LIN {X 0.078,Y -589.300,Z 1509.135,A 0.000,B 0.000,C 90.000,E1 60.205} C_DIS
LIN {X 0.071,Y -590.792,Z 1509.123,A 0.000,B 0.000,C 90.000,E1 58.074} C_DIS
LIN {X -0.260,Y -591.564,Z 1509.117,A 0.000,B 0.000,C 90.000,E1 57.041} C_DIS
LIN {X 0.336,Y -592.759,Z 1509.108,A 0.000,B 0.000,C 90.000,E1 55.388} C_DIS
LIN {X 0.156,Y -593.285,Z 1509.104,A 0.000,B 0.000,C 90.000,E1 54.609} C_DIS
LIN {X -0.185,Y -594.026,Z 1509.095,A 0.000,B 0.000,C 90.000,E1 53.050} C_DIS
LIN {X 0.067,Y -594.863,Z 1509.084,A 0.000,B 0.000,C 90.000,E1 51.170} C_DIS
LIN {X 0.249,Y -595.682,Z 1509.074,A 0.000,B 0.000,C 90.000,E1 49.299} C_DIS
LIN {X 0.240,Y -595.941,Z 1509.071,A 0.000,B 0.000,C 90.000,E1 48.771} C_DIS
LIN {X 0.220,Y -596.064,Z 1509.065,A 0.000,B 0.000,C 90.000,E1 47.715} C_DIS
LIN {X -0.242,Y -596.037,Z 1509.059,A 0.000,B 0.000,C 90.000,E1 46.701} C_DIS
LIN {X -0.293,Y -595.880,Z 1509.053,A 0.000,B 0.000,C 90.000,E1 45.648} C_DIS
LIN {X 0.106,Y -595.808,Z 1509.051,A 0.000,B 0.000,C 90.000,E1 45.081} C_DIS
LIN {X -0.170,Y -595.079,Z 1509.043,A 0.000,B 0.000,C 90.000,E1 43.785} C_DIS
LIN {X -0.010,Y -594.518,Z 1509.039,A 0.000,B 0.000,C 90.000,E1 42.975} C_DIS
LIN {X -0.054,Y -593.537,Z 1509.033,A 0.000,B 0.000,C 90.000,E1 41.919} C_DIS
LIN {X -0.103,Y -592.480,Z 1509.027,A 0.000,B 0.000,C 90.000,E1 40.862} C_DIS
LIN {X -0.164,Y -591.177,Z 1509.021,A 0.000,B 0.000,C 90.000,E1 39.806} C_DIS
LIN {X -0.249,Y -589.695,Z 1509.015,A 0.000,B 0.000,C 90.000,E1 38.749} C_DIS
LIN {X 0.097,Y -587.768,Z 1509.009,A 0.000,B 0.000,C 90.000,E1 37.649} C_DIS
LIN {X -0.136,Y -586.038,Z 1509.005,A 0.000,B 0.000,C 90.000,E1 36.870} C_DIS
LIN {X 0.248,Y -584.795,Z 1509.002,A 0.000,B 0.000,C 90.000,E1 36.297} C_DIS
LIN {X -0.195,Y -583.162,Z 1508.999,A 0.000,B 0.000,C 90.000,E1 35.804} C_DIS
LIN {X 0.165,Y -581.111,Z 1508.996,A 0.000,B 0.000,C 90.000,E1 35.231} C_DIS
LIN {X 0.256,Y -579.158,Z 1508.994,A 0.000,B 0.000,C 90.000,E1 34.818} C_DIS
LIN {X 0.092,Y -577.527,Z 1508.992,A 0.000,B 0.000,C 90.000,E1 34.565} C_DIS
LIN {X -0.139,Y -576.519,Z 1508.991,A 0.000,B 0.000,C 90.000,E1 34.452} C_DIS
LIN {X -0.224,Y -575.268,Z 1508.991,A 0.000,B 0.000,C 90.000,E1 34.326} C_DIS
LIN {X -0.308,Y -573.503,Z 1508.990,A 0.000,B 0.000,C 90.000,E1 34.199} C_DIS
LIN {X -0.047,Y -572.090,Z 1508.990,A 0.000,B 0.000,C 90.000,E1 34.119} C_DIS
LIN {X -0.068,Y -397.232,Z 1508.990,A 0.000,B 0.000,C 90.000,E1 34.119} C_DIS
LIN {X 0.195,Y -393.782,Z 1508.977,A 0.000,B 0.000,C 90.000,E1 31.799} C_DIS
LIN {X -0.045,Y -386.366,Z 1508.953,A 0.000,B 0.000,C 90.000,E1 27.564} C_DIS
LIN {X -0.081,Y -382.658,Z 1508.937,A 0.000,B 0.000,C 90.000,E1 24.695} C_DIS
LIN {X -0.148,Y -376.010,Z 1508.911,A 0.000,B 0.000,C 90.000,E1 19.993} C_DIS
LIN {X 0.069,Y -373.539,Z 1508.897,A 0.000,B 0.000,C 90.000,E1 17.402} C_DIS
LIN {X 0.108,Y -367.967,Z 1508.868,A 0.000,B 0.000,C 90.000,E1 12.243} C_DIS
LIN {X 0.126,Y -366.545,Z 1508.856,A 0.000,B 0.000,C 90.000,E1 10.018} C_DIS
LIN {X -0.161,Y -365.829,Z 1508.852,A 0.000,B 0.000,C 90.000,E1 9.321} C_DIS
LIN {X -0.146,Y -361.394,Z 1508.817,A 0.000,B 0.000,C 90.000,E1 2.980} C_DIS
LIN {X -0.055,Y -360.906,Z 1508.802,A 0.000,B 0.000,C 90.000,E1 0.344} C_DIS
LIN {X -0.092,Y -360.152,Z 1508.793,A 0.000,B 0.000,C 90.000,E1 358.682} C_DIS
LIN {X -0.053,Y -359.426,Z 1508.770,A 0.000,B 0.000,C 90.000,E1 354.546} C_DIS
LIN {X 0.070,Y -358.890,Z 1508.759,A 0.000,B 0.000,C 90.000,E1 352.648} C_DIS
LIN {X -0.020,Y -359.563,Z 1508.726,A 0.000,B 0.000,C 90.000,E1 346.645} C_DIS
LIN {X 0.001,Y -361.801,Z 1508.684,A 0.000,B 0.000,C 90.000,E1 339.135} C_DIS
LIN {X -0.154,Y -362.053,Z 1508.680,A 0.000,B 0.000,C 90.000,E1 338.411} C_DIS
LIN {X 0.189,Y -365.980,Z 1508.643,A 0.000,B 0.000,C 90.000,E1 331.641} C_DIS
LIN {X 0.029,Y -366.387,Z 1508.639,A 0.000,B 0.000,C 90.000,E1 330.923} C_DIS
LIN {X -0.031,Y -371.355,Z 1508.604,A 0.000,B 0.000,C 90.000,E1 324.642} C_DIS
LIN {X -0.043,Y -371.766,Z 1508.602,A 0.000,B 0.000,C 90.000,E1 324.276} C_DIS
LIN {X 0.013,Y -377.358,Z 1508.567,A 0.000,B 0.000,C 90.000,E1 318.038} C_DIS
LIN {X 0.012,Y -378.235,Z 1508.563,A 0.000,B 0.000,C 90.000,E1 317.310} C_DIS
LIN {X 0.002,Y -383.940,Z 1508.531,A 0.000,B 0.000,C 90.000,E1 311.515} C_DIS
LIN {X 0.088,Y -384.893,Z 1508.527,A 0.000,B 0.000,C 90.000,E1 310.782} C_DIS
LIN {X 0.262,Y -390.610,Z 1508.495,A 0.000,B 0.000,C 90.000,E1 305.025} C_DIS
LIN {X 0.106,Y -391.104,Z 1508.493,A 0.000,B 0.000,C 90.000,E1 304.692} C_DIS
LIN {X 0.022,Y -391.648,Z 1508.489,A 0.000,B 0.000,C 90.000,E1 303.992} C_DIS
LIN {X -0.080,Y -396.825,Z 1508.459,A 0.000,B 0.000,C 90.000,E1 298.693} C_DIS
LIN {X -0.210,Y -397.120,Z 1508.457,A 0.000,B 0.000,C 90.000,E1 298.359} C_DIS
LIN {X -0.055,Y -401.597,Z 1508.426,A 0.000,B 0.000,C 90.000,E1 292.717} C_DIS
LIN {X 0.222,Y -404.659,Z 1508.395,A 0.000,B 0.000,C 90.000,E1 287.094} C_DIS
LIN {X -0.079,Y -404.735,Z 1508.391,A 0.000,B 0.000,C 90.000,E1 286.441} C_DIS
LIN {X 0.214,Y -406.099,Z 1508.364,A 0.000,B 0.000,C 90.000,E1 281.535} C_DIS
LIN {X -0.176,Y -406.094,Z 1508.362,A 0.000,B 0.000,C 90.000,E1 281.243} C_DIS
LIN {X -0.097,Y -405.680,Z 1508.333,A 0.000,B 0.000,C 90.000,E1 276.024} C_DIS
LIN {X -0.165,Y -405.058,Z 1508.328,A 0.000,B 0.000,C 90.000,E1 274.992} C_DIS
LIN {X -0.060,Y -403.497,Z 1508.304,A 0.000,B 0.000,C 90.000,E1 270.802} C_DIS
LIN {X -0.092,Y -403.288,Z 1508.302,A 0.000,B 0.000,C 90.000,E1 270.458} C_DIS
LIN {X 0.091,Y -398.931,Z 1508.271,A 0.000,B 0.000,C 90.000,E1 264.837} C_DIS
LIN {X -0.040,Y -393.108,Z 1508.242,A 0.000,B 0.000,C 90.000,E1 259.567} C_DIS
LIN {X -0.079,Y -392.835,Z 1508.240,A 0.000,B 0.000,C 90.000,E1 259.218} C_DIS
LIN {X 0.034,Y -385.993,Z 1508.212,A 0.000,B 0.000,C 90.000,E1 254.212} C_DIS
LIN {X -0.026,Y -385.267,Z 1508.208,A 0.000,B 0.000,C 90.000,E1 253.504} C_DIS
LIN {X -0.004,Y -384.768,Z 1508.206,A 0.000,B 0.000,C 90.000,E1 253.142} C_DIS
LIN {X 0.221,Y -377.973,Z 1508.182,A 0.000,B 0.000,C 90.000,E1 248.773} C_DIS
LIN {X -0.044,Y -376.233,Z 1508.174,A 0.000,B 0.000,C 90.000,E1 247.358} C_DIS
LIN {X 0.057,Y -374.944,Z 1508.170,A 0.000,B 0.000,C 90.000,E1 246.613} C_DIS
LIN {X -0.208,Y -368.417,Z 1508.148,A 0.000,B 0.000,C 90.000,E1 242.615} C_DIS
LIN {X 0.097,Y -366.047,Z 1508.137,A 0.000,B 0.000,C 90.000,E1 240.717} C_DIS
LIN {X 0.004,Y -359.196,Z 1508.115,A 0.000,B 0.000,C 90.000,E1 236.628} C_DIS
LIN {X 0.021,Y -355.842,Z 1508.100,A 0.000,B 0.000,C 90.000,E1 233.989} C_DIS
LIN {X -0.173,Y -348.793,Z 1508.075,A 0.000,B 0.000,C 90.000,E1 229.461} C_DIS
LIN {X -0.097,Y -346.185,Z 1508.062,A 0.000,B 0.000,C 90.000,E1 227.148} C_DIS
LIN {X -0.088,Y -345.065,Z 1508.058,A 0.000,B 0.000,C 90.000,E1 226.377} C_DIS
LIN {X 0.094,Y -338.586,Z 1508.030,A 0.000,B 0.000,C 90.000,E1 221.310} C_DIS
LIN {X 0.094,Y -336.840,Z 1508.019,A 0.000,B 0.000,C 90.000,E1 219.358} C_DIS
LIN {X 0.014,Y -330.861,Z 1507.988,A 0.000,B 0.000,C 90.000,E1 213.865} C_DIS
LIN {X 0.149,Y -329.296,Z 1507.975,A 0.000,B 0.000,C 90.000,E1 211.465} C_DIS
LIN {X -0.154,Y -324.669,Z 1507.942,A 0.000,B 0.000,C 90.000,E1 205.540} C_DIS
LIN {X 0.174,Y -323.837,Z 1507.928,A 0.000,B 0.000,C 90.000,E1 203.078} C_DIS
LIN {X -0.017,Y -321.124,Z 1507.881,A 0.000,B 0.000,C 90.000,E1 194.662} C_DIS
LIN {X 0.138,Y -320.932,Z 1507.877,A 0.000,B 0.000,C 90.000,E1 193.828} C_DIS
LIN {X -0.076,Y -321.562,Z 1507.832,A 0.000,B 0.000,C 90.000,E1 185.796} C_DIS
LIN {X -0.143,Y -324.415,Z 1507.790,A 0.000,B 0.000,C 90.000,E1 178.165} C_DIS
LIN {X -0.141,Y -325.376,Z 1507.783,A 0.000,B 0.000,C 90.000,E1 176.963} C_DIS
LIN {X -0.100,Y -329.112,Z 1507.750,A 0.000,B 0.000,C 90.000,E1 170.971} C_DIS
LIN {X 0.061,Y -334.260,Z 1507.726,A 0.000,B 0.000,C 90.000,E1 166.589} C_DIS
LIN {X 0.067,Y -335.488,Z 1507.719,A 0.000,B 0.000,C 90.000,E1 165.408} C_DIS
LIN {X 0.143,Y -340.932,Z 1507.695,A 0.000,B 0.000,C 90.000,E1 161.094} C_DIS
LIN {X -0.172,Y -342.138,Z 1507.691,A 0.000,B 0.000,C 90.000,E1 160.369} C_DIS
LIN {X -0.058,Y -347.939,Z 1507.667,A 0.000,B 0.000,C 90.000,E1 156.102} C_DIS
LIN {X -0.081,Y -354.259,Z 1507.648,A 0.000,B 0.000,C 90.000,E1 152.666} C_DIS
LIN {X -0.222,Y -361.406,Z 1507.625,A 0.000,B 0.000,C 90.000,E1 148.535} C_DIS
LIN {X 0.065,Y -368.758,Z 1507.606,A 0.000,B 0.000,C 90.000,E1 145.135} C_DIS
LIN {X 0.115,Y -371.571,Z 1507.598,A 0.000,B 0.000,C 90.000,E1 143.623} C_DIS
LIN {X 0.116,Y -532.806,Z 1507.598,A 0.000,B 0.000,C 90.000,E1 143.623} C_DIS
LIN {X 0.022,Y -533.281,Z 1507.598,A 0.000,B 0.000,C 90.000,E1 143.623} C_DIS
LIN {X -0.004,Y -535.709,Z 1507.597,A 0.000,B 0.000,C 90.000,E1 143.463} C_DIS
LIN {X 0.080,Y -537.063,Z 1507.596,A 0.000,B 0.000,C 90.000,E1 143.290} C_DIS
LIN {X 0.083,Y -538.840,Z 1507.595,A 0.000,B 0.000,C 90.000,E1 143.004} C_DIS
LIN {X 0.094,Y -540.246,Z 1507.593,A 0.000,B 0.000,C 90.000,E1 142.718} C_DIS
LIN {X 0.111,Y -541.397,Z 1507.591,A 0.000,B 0.000,C 90.000,E1 142.431} C_DIS
LIN {X -0.275,Y -543.302,Z 1507.588,A 0.000,B 0.000,C 90.000,E1 141.904} C_DIS
LIN {X -0.218,Y -544.761,Z 1507.585,A 0.000,B 0.000,C 90.000,E1 141.331} C_DIS
LIN {X 0.192,Y -545.888,Z 1507.582,A 0.000,B 0.000,C 90.000,E1 140.723} C_DIS
LIN {X -0.075,Y -547.779,Z 1507.576,A 0.000,B 0.000,C 90.000,E1 139.622} C_DIS
LIN {X 0.035,Y -549.509,Z 1507.569,A 0.000,B 0.000,C 90.000,E1 138.485} C_DIS
LIN {X 0.179,Y -551.445,Z 1507.562,A 0.000,B 0.000,C 90.000,E1 137.067} C_DIS
LIN {X 0.289,Y -552.461,Z 1507.557,A 0.000,B 0.000,C 90.000,E1 136.215} C_DIS
LIN {X 0.092,Y -554.032,Z 1507.549,A 0.000,B 0.000,C 90.000,E1 134.838} C_DIS
LIN {X 0.266,Y -555.081,Z 1507.543,A 0.000,B 0.000,C 90.000,E1 133.704} C_DIS
LIN {X 0.070,Y -556.027,Z 1507.537,A 0.000,B 0.000,C 90.000,E1 132.609} C_DIS
LIN {X -0.045,Y -557.038,Z 1507.529,A 0.000,B 0.000,C 90.000,E1 131.229} C_DIS
LIN {X -0.145,Y -557.939,Z 1507.521,A 0.000,B 0.000,C 90.000,E1 129.850} C_DIS
LIN {X -0.074,Y -558.896,Z 1507.512,A 0.000,B 0.000,C 90.000,E1 128.177} C_DIS
LIN {X -0.071,Y -559.585,Z 1507.504,A 0.000,B 0.000,C 90.000,E1 126.790} C_DIS
LIN {X -0.035,Y -559.941,Z 1507.498,A 0.000,B 0.000,C 90.000,E1 125.678} C_DIS
LIN {X 0.107,Y -560.169,Z 1507.491,A 0.000,B 0.000,C 90.000,E1 124.278} C_DIS
LIN {X 0.158,Y -560.188,Z 1507.484,A 0.000,B 0.000,C 90.000,E1 123.166} C_DIS
LIN {X -0.007,Y -560.169,Z 1507.469,A 0.000,B 0.000,C 90.000,E1 120.413} C_DIS
LIN {X 0.015,Y -560.435,Z 1507.461,A 0.000,B 0.000,C 90.000,E1 119.027} C_DIS
LIN {X -0.170,Y -560.716,Z 1507.452,A 0.000,B 0.000,C 90.000,E1 117.385} C_DIS
LIN {X -0.117,Y -561.052,Z 1507.443,A 0.000,B 0.000,C 90.000,E1 115.720} C_DIS
LIN {X -0.299,Y -561.384,Z 1507.434,A 0.000,B 0.000,C 90.000,E1 114.079} C_DIS
LIN {X -0.077,Y -561.613,Z 1507.427,A 0.000,B 0.000,C 90.000,E1 112.950} C_DIS
LIN {X 0.042,Y -561.971,Z 1507.418,A 0.000,B 0.000,C 90.000,E1 111.280} C_DIS
LIN {X 0.280,Y -562.341,Z 1507.408,A 0.000,B 0.000,C 90.000,E1 109.322} C_DIS
LIN {X 0.163,Y -562.713,Z 1507.397,A 0.000,B 0.000,C 90.000,E1 107.402} C_DIS
LIN {X 0.144,Y -563.056,Z 1507.389,A 0.000,B 0.000,C 90.000,E1 106.024} C_DIS
LIN {X 0.276,Y -563.533,Z 1507.380,A 0.000,B 0.000,C 90.000,E1 104.356} C_DIS
LIN {X -0.243,Y -564.061,Z 1507.369,A 0.000,B 0.000,C 90.000,E1 102.479} C_DIS
LIN {X 0.033,Y -564.577,Z 1507.362,A 0.000,B 0.000,C 90.000,E1 101.074} C_DIS
LIN {X -0.008,Y -565.395,Z 1507.351,A 0.000,B 0.000,C 90.000,E1 99.151} C_DIS
LIN {X 0.015,Y -565.835,Z 1507.345,A 0.000,B 0.000,C 90.000,E1 98.049} C_DIS
LIN {X -0.265,Y -566.579,Z 1507.336,A 0.000,B 0.000,C 90.000,E1 96.429} C_DIS
LIN {X 0.183,Y -567.767,Z 1507.323,A 0.000,B 0.000,C 90.000,E1 94.188} C_DIS
LIN {X -0.174,Y -568.625,Z 1507.314,A 0.000,B 0.000,C 90.000,E1 92.579} C_DIS
LIN {X -0.103,Y -569.426,Z 1507.307,A 0.000,B 0.000,C 90.000,E1 91.203} C_DIS
LIN {X 0.100,Y -570.363,Z 1507.298,A 0.000,B 0.000,C 90.000,E1 89.542} C_DIS
LIN {X -0.234,Y -571.389,Z 1507.288,A 0.000,B 0.000,C 90.000,E1 87.936} C_DIS
LIN {X 0.155,Y -572.507,Z 1507.278,A 0.000,B 0.000,C 90.000,E1 85.988} C_DIS
LIN {X -0.060,Y -573.547,Z 1507.269,A 0.000,B 0.000,C 90.000,E1 84.375} C_DIS
LIN {X 0.273,Y -575.185,Z 1507.255,A 0.000,B 0.000,C 90.000,E1 81.894} C_DIS
LIN {X -0.172,Y -576.525,Z 1507.245,A 0.000,B 0.000,C 90.000,E1 80.038} C_DIS
LIN {X 0.076,Y -578.001,Z 1507.234,A 0.000,B 0.000,C 90.000,E1 78.117} C_DIS
LIN {X -0.181,Y -579.242,Z 1507.225,A 0.000,B 0.000,C 90.000,E1 76.520} C_DIS
LIN {X 0.163,Y -580.391,Z 1507.216,A 0.000,B 0.000,C 90.000,E1 74.866} C_DIS
LIN {X 0.081,Y -581.159,Z 1507.210,A 0.000,B 0.000,C 90.000,E1 73.795} C_DIS
LIN {X -0.162,Y -581.935,Z 1507.203,A 0.000,B 0.000,C 90.000,E1 72.472} C_DIS
LIN {X -0.235,Y -582.547,Z 1507.197,A 0.000,B 0.000,C 90.000,E1 71.402} C_DIS
LIN {X 0.131,Y -583.524,Z 1507.188,A 0.000,B 0.000,C 90.000,E1 69.752} C_DIS
LIN {X -0.155,Y -584.537,Z 1507.177,A 0.000,B 0.000,C 90.000,E1 67.901} C_DIS
LIN {X 0.110,Y -585.580,Z 1507.167,A 0.000,B 0.000,C 90.000,E1 65.997} C_DIS
LIN {X -0.086,Y -586.594,Z 1507.158,A 0.000,B 0.000,C 90.000,E1 64.409} C_DIS
LIN {X 0.009,Y -587.682,Z 1507.149,A 0.000,B 0.000,C 90.000,E1 62.794} C_DIS
LIN {X 0.244,Y -588.688,Z 1507.141,A 0.000,B 0.000,C 90.000,E1 61.435} C_DIS
LIN {X -0.026,Y -589.641,Z 1507.134,A 0.000,B 0.000,C 90.000,E1 60.127} C_DIS
LIN {X -0.098,Y -590.746,Z 1507.125,A 0.000,B 0.000,C 90.000,E1 58.535} C_DIS
LIN {X 0.069,Y -591.569,Z 1507.119,A 0.000,B 0.000,C 90.000,E1 57.454} C_DIS
LIN {X -0.039,Y -592.579,Z 1507.112,A 0.000,B 0.000,C 90.000,E1 56.135} C_DIS
LIN {X -0.123,Y -593.527,Z 1507.104,A 0.000,B 0.000,C 90.000,E1 54.815} C_DIS
LIN {X 0.019,Y -594.291,Z 1507.096,A 0.000,B 0.000,C 90.000,E1 53.210} C_DIS
LIN {X -0.174,Y -594.899,Z 1507.088,A 0.000,B 0.000,C 90.000,E1 51.904} C_DIS
LIN {X 0.242,Y -595.585,Z 1507.079,A 0.000,B 0.000,C 90.000,E1 50.275} C_DIS
LIN {X 0.225,Y -596.091,Z 1507.074,A 0.000,B 0.000,C 90.000,E1 49.218} C_DIS
LIN {X 0.218,Y -596.358,Z 1507.071,A 0.000,B 0.000,C 90.000,E1 48.690} C_DIS
LIN {X -0.018,Y -596.431,Z 1507.063,A 0.000,B 0.000,C 90.000,E1 47.391} C_DIS
LIN {X 0.147,Y -596.343,Z 1507.056,A 0.000,B 0.000,C 90.000,E1 46.053} C_DIS
LIN {X 0.104,Y -596.145,Z 1507.050,A 0.000,B 0.000,C 90.000,E1 45.000} C_DIS
LIN {X -0.166,Y -595.418,Z 1507.043,A 0.000,B 0.000,C 90.000,E1 43.704} C_DIS
LIN {X 0.205,Y -594.612,Z 1507.037,A 0.000,B 0.000,C 90.000,E1 42.609} C_DIS
LIN {X -0.064,Y -593.376,Z 1507.030,A 0.000,B 0.000,C 90.000,E1 41.310} C_DIS
LIN {X 0.096,Y -591.808,Z 1507.022,A 0.000,B 0.000,C 90.000,E1 39.967} C_DIS
LIN {X -0.184,Y -590.801,Z 1507.018,A 0.000,B 0.000,C 90.000,E1 39.197} C_DIS
LIN {X 0.180,Y -589.016,Z 1507.012,A 0.000,B 0.000,C 90.000,E1 38.096} C_DIS
LIN {X 0.119,Y -588.052,Z 1507.009,A 0.000,B 0.000,C 90.000,E1 37.569} C_DIS
LIN {X 0.080,Y -585.758,Z 1507.003,A 0.000,B 0.000,C 90.000,E1 36.503} C_DIS
LIN {X -0.171,Y -583.729,Z 1506.998,A 0.000,B 0.000,C 90.000,E1 35.724} C_DIS
LIN {X -0.143,Y -582.106,Z 1506.995,A 0.000,B 0.000,C 90.000,E1 35.185} C_DIS
LIN {X 0.208,Y -580.035,Z 1506.992,A 0.000,B 0.000,C 90.000,E1 34.612} C_DIS
LIN {X 0.049,Y -578.743,Z 1506.991,A 0.000,B 0.000,C 90.000,E1 34.358} C_DIS
LIN {X -0.265,Y -577.195,Z 1506.990,A 0.000,B 0.000,C 90.000,E1 34.119} C_DIS
LIN {X -0.108,Y -575.301,Z 1506.988,A 0.000,B 0.000,C 90.000,E1 33.833} C_DIS
LIN {X -0.194,Y -574.077,Z 1506.987,A 0.000,B 0.000,C 90.000,E1 33.706} C_DIS
LIN {X 0.238,Y -572.125,Z 1506.986,A 0.000,B 0.000,C 90.000,E1 33.499} C_DIS
LIN {X 0.056,Y -570.741,Z 1506.986,A 0.000,B 0.000,C 90.000,E1 33.452} C_DIS
LIN {X -0.073,Y -570.070,Z 1506.986,A 0.000,B 0.000,C 90.000,E1 33.452} C_DIS
LIN {X -0.081,Y -396.149,Z 1506.986,A 0.000,B 0.000,C 90.000,E1 33.452} C_DIS
LIN {X 0.127,Y -393.881,Z 1506.977,A 0.000,B 0.000,C 90.000,E1 31.878} C_DIS
LIN {X -0.096,Y -386.468,Z 1506.953,A 0.000,B 0.000,C 90.000,E1 27.641} C_DIS
LIN {X -0.119,Y -382.777,Z 1506.938,A 0.000,B 0.000,C 90.000,E1 24.771} C_DIS
LIN {X -0.164,Y -376.089,Z 1506.911,A 0.000,B 0.000,C 90.000,E1 20.066} C_DIS
LIN {X 0.178,Y -373.622,Z 1506.897,A 0.000,B 0.000,C 90.000,E1 17.457} C_DIS
LIN {X -0.149,Y -368.023,Z 1506.869,A 0.000,B 0.000,C 90.000,E1 12.355} C_DIS
LIN {X 0.084,Y -366.316,Z 1506.854,A 0.000,B 0.000,C 90.000,E1 9.726} C_DIS
LIN {X -0.037,Y -361.707,Z 1506.821,A 0.000,B 0.000,C 90.000,E1 3.784} C_DIS
LIN {X 0.044,Y -360.909,Z 1506.802,A 0.000,B 0.000,C 90.000,E1 0.401} C_DIS
LIN {X 0.137,Y -360.684,Z 1506.799,A 0.000,B 0.000,C 90.000,E1 359.771} C_DIS
LIN {X -0.053,Y -359.426,Z 1506.770,A 0.000,B 0.000,C 90.000,E1 354.546} C_DIS
LIN {X 0.070,Y -358.890,Z 1506.759,A 0.000,B 0.000,C 90.000,E1 352.648} C_DIS
LIN {X -0.020,Y -359.563,Z 1506.726,A 0.000,B 0.000,C 90.000,E1 346.645} C_DIS
LIN {X 0.001,Y -361.801,Z 1506.684,A 0.000,B 0.000,C 90.000,E1 339.135} C_DIS
LIN {X -0.154,Y -362.053,Z 1506.680,A 0.000,B 0.000,C 90.000,E1 338.411} C_DIS
LIN {X 0.189,Y -365.980,Z 1506.643,A 0.000,B 0.000,C 90.000,E1 331.641} C_DIS
LIN {X 0.029,Y -366.387,Z 1506.639,A 0.000,B 0.000,C 90.000,E1 330.923} C_DIS
LIN {X -0.031,Y -371.355,Z 1506.604,A 0.000,B 0.000,C 90.000,E1 324.642} C_DIS
LIN {X -0.043,Y -371.766,Z 1506.602,A 0.000,B 0.000,C 90.000,E1 324.276} C_DIS
LIN {X 0.013,Y -377.358,Z 1506.567,A 0.000,B 0.000,C 90.000,E1 318.038} C_DIS
LIN {X 0.012,Y -378.235,Z 1506.563,A 0.000,B 0.000,C 90.000,E1 317.310} C_DIS
LIN {X 0.002,Y -383.940,Z 1506.531,A 0.000,B 0.000,C 90.000,E1 311.515} C_DIS
LIN {X 0.088,Y -384.893,Z 1506.527,A 0.000,B 0.000,C 90.000,E1 310.782} C_DIS
LIN {X 0.262,Y -390.610,Z 1506.495,A 0.000,B 0.000,C 90.000,E1 305.025} C_DIS
LIN {X 0.106,Y -391.104,Z 1506.493,A 0.000,B 0.000,C 90.000,E1 304.692} C_DIS
LIN {X 0.022,Y -391.648,Z 1506.489,A 0.000,B 0.000,C 90.000,E1 303.992} C_DIS
LIN {X -0.080,Y -396.825,Z 1506.459,A 0.000,B 0.000,C 90.000,E1 298.693} C_DIS
LIN {X -0.210,Y -397.120,Z 1506.457,A 0.000,B 0.000,C 90.000,E1 298.359} C_DIS
LIN {X -0.055,Y -401.597,Z 1506.426,A 0.000,B 0.000,C 90.000,E1 292.717} C_DIS
LIN {X 0.222,Y -404.659,Z 1506.395,A 0.000,B 0.000,C 90.000,E1 287.094} C_DIS
LIN {X -0.079,Y -404.735,Z 1506.391,A 0.000,B 0.000,C 90.000,E1 286.441} C_DIS
LIN {X 0.214,Y -406.099,Z 1506.364,A 0.000,B 0.000,C 90.000,E1 281.535} C_DIS
LIN {X -0.176,Y -406.094,Z 1506.362,A 0.000,B 0.000,C 90.000,E1 281.243} C_DIS
LIN {X -0.097,Y -405.680,Z 1506.333,A 0.000,B 0.000,C 90.000,E1 276.024} C_DIS
LIN {X -0.165,Y -405.058,Z 1506.328,A 0.000,B 0.000,C 90.000,E1 274.992} C_DIS
LIN {X -0.060,Y -403.497,Z 1506.304,A 0.000,B 0.000,C 90.000,E1 270.802} C_DIS
LIN {X -0.092,Y -403.288,Z 1506.302,A 0.000,B 0.000,C 90.000,E1 270.458} C_DIS
LIN {X 0.091,Y -398.931,Z 1506.271,A 0.000,B 0.000,C 90.000,E1 264.837} C_DIS
LIN {X -0.040,Y -393.108,Z 1506.242,A 0.000,B 0.000,C 90.000,E1 259.567} C_DIS
LIN {X -0.079,Y -392.835,Z 1506.240,A 0.000,B 0.000,C 90.000,E1 259.218} C_DIS
LIN {X 0.034,Y -385.993,Z 1506.212,A 0.000,B 0.000,C 90.000,E1 254.212} C_DIS
LIN {X -0.026,Y -385.267,Z 1506.208,A 0.000,B 0.000,C 90.000,E1 253.504} C_DIS
LIN {X -0.004,Y -384.768,Z 1506.206,A 0.000,B 0.000,C 90.000,E1 253.142} C_DIS
LIN {X 0.221,Y -377.973,Z 1506.182,A 0.000,B 0.000,C 90.000,E1 248.773} C_DIS
LIN {X -0.044,Y -376.233,Z 1506.174,A 0.000,B 0.000,C 90.000,E1 247.358} C_DIS
LIN {X 0.057,Y -374.944,Z 1506.170,A 0.000,B 0.000,C 90.000,E1 246.613} C_DIS
LIN {X -0.208,Y -368.417,Z 1506.148,A 0.000,B 0.000,C 90.000,E1 242.615} C_DIS
LIN {X 0.097,Y -366.047,Z 1506.137,A 0.000,B 0.000,C 90.000,E1 240.717} C_DIS
LIN {X 0.004,Y -359.196,Z 1506.115,A 0.000,B 0.000,C 90.000,E1 236.628} C_DIS
LIN {X 0.021,Y -355.842,Z 1506.100,A 0.000,B 0.000,C 90.000,E1 233.989} C_DIS
LIN {X -0.173,Y -348.793,Z 1506.075,A 0.000,B 0.000,C 90.000,E1 229.461} C_DIS
LIN {X -0.097,Y -346.185,Z 1506.062,A 0.000,B 0.000,C 90.000,E1 227.148} C_DIS
LIN {X -0.088,Y -345.065,Z 1506.058,A 0.000,B 0.000,C 90.000,E1 226.377} C_DIS
LIN {X 0.094,Y -338.586,Z 1506.030,A 0.000,B 0.000,C 90.000,E1 221.310} C_DIS
LIN {X 0.094,Y -336.840,Z 1506.019,A 0.000,B 0.000,C 90.000,E1 219.358} C_DIS
LIN {X 0.014,Y -330.861,Z 1505.988,A 0.000,B 0.000,C 90.000,E1 213.865} C_DIS
LIN {X 0.149,Y -329.296,Z 1505.975,A 0.000,B 0.000,C 90.000,E1 211.465} C_DIS
LIN {X -0.154,Y -324.669,Z 1505.942,A 0.000,B 0.000,C 90.000,E1 205.540} C_DIS
LIN {X 0.174,Y -323.837,Z 1505.928,A 0.000,B 0.000,C 90.000,E1 203.078} C_DIS
LIN {X -0.017,Y -321.124,Z 1505.881,A 0.000,B 0.000,C 90.000,E1 194.662} C_DIS
LIN {X 0.138,Y -320.932,Z 1505.877,A 0.000,B 0.000,C 90.000,E1 193.828} C_DIS
LIN {X -0.076,Y -321.562,Z 1505.832,A 0.000,B 0.000,C 90.000,E1 185.796} C_DIS
LIN {X -0.143,Y -324.415,Z 1505.790,A 0.000,B 0.000,C 90.000,E1 178.165} C_DIS
LIN {X -0.141,Y -325.376,Z 1505.783,A 0.000,B 0.000,C 90.000,E1 176.963} C_DIS
LIN {X -0.100,Y -329.112,Z 1505.750,A 0.000,B 0.000,C 90.000,E1 170.971} C_DIS
LIN {X 0.061,Y -334.260,Z 1505.726,A 0.000,B 0.000,C 90.000,E1 166.589} C_DIS
LIN {X 0.067,Y -335.488,Z 1505.719,A 0.000,B 0.000,C 90.000,E1 165.408} C_DIS
LIN {X 0.143,Y -340.932,Z 1505.695,A 0.000,B 0.000,C 90.000,E1 161.094} C_DIS
LIN {X -0.172,Y -342.138,Z 1505.691,A 0.000,B 0.000,C 90.000,E1 160.369} C_DIS
LIN {X -0.058,Y -347.939,Z 1505.667,A 0.000,B 0.000,C 90.000,E1 156.102} C_DIS
LIN {X -0.081,Y -354.259,Z 1505.648,A 0.000,B 0.000,C 90.000,E1 152.666} C_DIS
LIN {X -0.222,Y -361.406,Z 1505.625,A 0.000,B 0.000,C 90.000,E1 148.535} C_DIS
LIN {X 0.065,Y -368.758,Z 1505.606,A 0.000,B 0.000,C 90.000,E1 145.135} C_DIS
LIN {X -0.087,Y -370.134,Z 1505.602,A 0.000,B 0.000,C 90.000,E1 144.402} C_DIS
LIN {X -0.175,Y -531.396,Z 1505.602,A 0.000,B 0.000,C 90.000,E1 144.402} C_DIS
LIN {X 0.129,Y -534.351,Z 1505.601,A 0.000,B 0.000,C 90.000,E1 144.196} C_DIS
LIN {X 0.001,Y -535.820,Z 1505.600,A 0.000,B 0.000,C 90.000,E1 144.036} C_DIS
LIN {X 0.001,Y -537.611,Z 1505.599,A 0.000,B 0.000,C 90.000,E1 143.749} C_DIS
LIN {X -0.144,Y -539.689,Z 1505.596,A 0.000,B 0.000,C 90.000,E1 143.336} C_DIS
LIN {X -0.282,Y -541.330,Z 1505.594,A 0.000,B 0.000,C 90.000,E1 142.924} C_DIS
LIN {X 0.093,Y -543.050,Z 1505.591,A 0.000,B 0.000,C 90.000,E1 142.316} C_DIS
LIN {X 0.154,Y -544.417,Z 1505.588,A 0.000,B 0.000,C 90.000,E1 141.743} C_DIS
LIN {X 0.257,Y -546.015,Z 1505.583,A 0.000,B 0.000,C 90.000,E1 140.884} C_DIS
LIN {X -0.010,Y -547.884,Z 1505.577,A 0.000,B 0.000,C 90.000,E1 139.784} C_DIS
LIN {X 0.099,Y -549.643,Z 1505.570,A 0.000,B 0.000,C 90.000,E1 138.647} C_DIS
LIN {X 0.242,Y -551.571,Z 1505.563,A 0.000,B 0.000,C 90.000,E1 137.229} C_DIS
LIN {X -0.001,Y -552.907,Z 1505.556,A 0.000,B 0.000,C 90.000,E1 136.134} C_DIS
LIN {X 0.158,Y -554.181,Z 1505.550,A 0.000,B 0.000,C 90.000,E1 135.000} C_DIS
LIN {X -0.011,Y -555.461,Z 1505.542,A 0.000,B 0.000,C 90.000,E1 133.623} C_DIS
LIN {X -0.203,Y -556.416,Z 1505.536,A 0.000,B 0.000,C 90.000,E1 132.528} C_DIS
LIN {X -0.312,Y -557.364,Z 1505.528,A 0.000,B 0.000,C 90.000,E1 131.148} C_DIS
LIN {X 0.020,Y -558.262,Z 1505.521,A 0.000,B 0.000,C 90.000,E1 129.725} C_DIS
LIN {X -0.334,Y -559.111,Z 1505.511,A 0.000,B 0.000,C 90.000,E1 128.096} C_DIS
LIN {X 0.119,Y -559.794,Z 1505.504,A 0.000,B 0.000,C 90.000,E1 126.664} C_DIS
LIN {X -0.293,Y -560.099,Z 1505.498,A 0.000,B 0.000,C 90.000,E1 125.598} C_DIS
LIN {X 0.073,Y -560.247,Z 1505.491,A 0.000,B 0.000,C 90.000,E1 124.452} C_DIS
LIN {X 0.028,Y -560.279,Z 1505.487,A 0.000,B 0.000,C 90.000,E1 123.627} C_DIS
LIN {X -0.144,Y -560.192,Z 1505.472,A 0.000,B 0.000,C 90.000,E1 120.875} C_DIS
LIN {X -0.054,Y -560.461,Z 1505.462,A 0.000,B 0.000,C 90.000,E1 119.205} C_DIS
LIN {X 0.252,Y -560.734,Z 1505.453,A 0.000,B 0.000,C 90.000,E1 117.513} C_DIS
LIN {X 0.305,Y -561.062,Z 1505.444,A 0.000,B 0.000,C 90.000,E1 115.848} C_DIS
LIN {X 0.125,Y -561.376,Z 1505.435,A 0.000,B 0.000,C 90.000,E1 114.207} C_DIS
LIN {X 0.146,Y -561.681,Z 1505.427,A 0.000,B 0.000,C 90.000,E1 112.823} C_DIS
LIN {X 0.061,Y -562.058,Z 1505.418,A 0.000,B 0.000,C 90.000,E1 111.173} C_DIS
LIN {X 0.185,Y -562.367,Z 1505.408,A 0.000,B 0.000,C 90.000,E1 109.504} C_DIS
LIN {X 0.067,Y -562.769,Z 1505.398,A 0.000,B 0.000,C 90.000,E1 107.583} C_DIS
LIN {X -0.186,Y -563.168,Z 1505.389,A 0.000,B 0.000,C 90.000,E1 105.953} C_DIS
LIN {X -0.201,Y -563.644,Z 1505.379,A 0.000,B 0.000,C 90.000,E1 104.300} C_DIS
LIN {X -0.204,Y -564.138,Z 1505.370,A 0.000,B 0.000,C 90.000,E1 102.647} C_DIS
LIN {X 0.229,Y -564.724,Z 1505.361,A 0.000,B 0.000,C 90.000,E1 100.950} C_DIS
LIN {X 0.180,Y -565.562,Z 1505.350,A 0.000,B 0.000,C 90.000,E1 99.029} C_DIS
LIN {X -0.109,Y -566.238,Z 1505.341,A 0.000,B 0.000,C 90.000,E1 97.409} C_DIS
LIN {X 0.111,Y -567.003,Z 1505.332,A 0.000,B 0.000,C 90.000,E1 95.739} C_DIS
LIN {X -0.261,Y -567.976,Z 1505.323,A 0.000,B 0.000,C 90.000,E1 94.131} C_DIS
LIN {X -0.168,Y -568.698,Z 1505.315,A 0.000,B 0.000,C 90.000,E1 92.751} C_DIS
LIN {X -0.097,Y -569.542,Z 1505.308,A 0.000,B 0.000,C 90.000,E1 91.375} C_DIS
LIN {X -0.199,Y -570.833,Z 1505.296,A 0.000,B 0.000,C 90.000,E1 89.198} C_DIS
LIN {X 0.046,Y -571.849,Z 1505.286,A 0.000,B 0.000,C 90.000,E1 87.535} C_DIS
LIN {X -0.226,Y -572.813,Z 1505.277,A 0.000,B 0.000,C 90.000,E1 85.927} C_DIS
LIN {X 0.095,Y -573.881,Z 1505.268,A 0.000,B 0.000,C 90.000,E1 84.261} C_DIS
LIN {X 0.312,Y -575.331,Z 1505.256,A 0.000,B 0.000,C 90.000,E1 82.064} C_DIS
LIN {X -0.178,Y -576.087,Z 1505.250,A 0.000,B 0.000,C 90.000,E1 81.027} C_DIS
LIN {X -0.153,Y -577.301,Z 1505.241,A 0.000,B 0.000,C 90.000,E1 79.398} C_DIS
LIN {X 0.014,Y -578.582,Z 1505.232,A 0.000,B 0.000,C 90.000,E1 77.757} C_DIS
LIN {X 0.206,Y -579.812,Z 1505.223,A 0.000,B 0.000,C 90.000,E1 76.117} C_DIS
LIN {X -0.010,Y -580.949,Z 1505.214,A 0.000,B 0.000,C 90.000,E1 74.519} C_DIS
LIN {X -0.093,Y -581.670,Z 1505.208,A 0.000,B 0.000,C 90.000,E1 73.449} C_DIS
LIN {X -0.337,Y -582.429,Z 1505.201,A 0.000,B 0.000,C 90.000,E1 72.127} C_DIS
LIN {X 0.087,Y -583.733,Z 1505.189,A 0.000,B 0.000,C 90.000,E1 69.934} C_DIS
LIN {X 0.131,Y -584.722,Z 1505.178,A 0.000,B 0.000,C 90.000,E1 68.050} C_DIS
LIN {X 0.084,Y -585.771,Z 1505.168,A 0.000,B 0.000,C 90.000,E1 66.177} C_DIS
LIN {X -0.219,Y -586.957,Z 1505.157,A 0.000,B 0.000,C 90.000,E1 64.332} C_DIS
LIN {X 0.143,Y -588.038,Z 1505.148,A 0.000,B 0.000,C 90.000,E1 62.692} C_DIS
LIN {X -0.033,Y -588.884,Z 1505.142,A 0.000,B 0.000,C 90.000,E1 61.641} C_DIS
LIN {X -0.122,Y -589.982,Z 1505.134,A 0.000,B 0.000,C 90.000,E1 60.049} C_DIS
LIN {X -0.377,Y -590.918,Z 1505.126,A 0.000,B 0.000,C 90.000,E1 58.742} C_DIS
LIN {X -0.006,Y -591.914,Z 1505.119,A 0.000,B 0.000,C 90.000,E1 57.375} C_DIS
LIN {X 0.389,Y -592.971,Z 1505.111,A 0.000,B 0.000,C 90.000,E1 56.008} C_DIS
LIN {X 0.089,Y -593.759,Z 1505.105,A 0.000,B 0.000,C 90.000,E1 54.975} C_DIS
LIN {X 0.362,Y -594.430,Z 1505.098,A 0.000,B 0.000,C 90.000,E1 53.623} C_DIS
LIN {X -0.187,Y -595.059,Z 1505.091,A 0.000,B 0.000,C 90.000,E1 52.351} C_DIS
LIN {X -0.007,Y -595.886,Z 1505.080,A 0.000,B 0.000,C 90.000,E1 50.481} C_DIS
LIN {X -0.404,Y -596.411,Z 1505.075,A 0.000,B 0.000,C 90.000,E1 49.461} C_DIS
LIN {X 0.206,Y -596.763,Z 1505.070,A 0.000,B 0.000,C 90.000,E1 48.609} C_DIS
LIN {X -0.023,Y -596.786,Z 1505.063,A 0.000,B 0.000,C 90.000,E1 47.310} C_DIS
LIN {X -0.072,Y -596.632,Z 1505.054,A 0.000,B 0.000,C 90.000,E1 45.729} C_DIS
LIN {X 0.331,Y -596.583,Z 1505.051,A 0.000,B 0.000,C 90.000,E1 45.162} C_DIS
LIN {X 0.070,Y -595.895,Z 1505.044,A 0.000,B 0.000,C 90.000,E1 43.866} C_DIS
LIN {X 0.011,Y -595.177,Z 1505.038,A 0.000,B 0.000,C 90.000,E1 42.813} C_DIS
LIN {X 0.189,Y -593.968,Z 1505.031,A 0.000,B 0.000,C 90.000,E1 41.472} C_DIS
LIN {X -0.065,Y -593.046,Z 1505.026,A 0.000,B 0.000,C 90.000,E1 40.701} C_DIS
LIN {X -0.159,Y -591.099,Z 1505.017,A 0.000,B 0.000,C 90.000,E1 39.116} C_DIS
LIN {X 0.051,Y -588.881,Z 1505.010,A 0.000,B 0.000,C 90.000,E1 37.764} C_DIS
LIN {X 0.111,Y -586.036,Z 1505.002,A 0.000,B 0.000,C 90.000,E1 36.423} C_DIS
LIN {X -0.111,Y -582.618,Z 1504.995,A 0.000,B 0.000,C 90.000,E1 35.105} C_DIS
LIN {X 0.242,Y -580.949,Z 1504.992,A 0.000,B 0.000,C 90.000,E1 34.532} C_DIS
LIN {X 0.255,Y -578.706,Z 1504.989,A 0.000,B 0.000,C 90.000,E1 33.992} C_DIS
LIN {X -0.146,Y -576.569,Z 1504.987,A 0.000,B 0.000,C 90.000,E1 33.627} C_DIS
LIN {X -0.311,Y -574.914,Z 1504.985,A 0.000,B 0.000,C 90.000,E1 33.372} C_DIS
LIN {X -0.165,Y -572.843,Z 1504.984,A 0.000,B 0.000,C 90.000,E1 33.086} C_DIS
LIN {X 0.253,Y -571.002,Z 1504.983,A 0.000,B 0.000,C 90.000,E1 32.880} C_DIS
LIN {X -0.124,Y -569.534,Z 1504.982,A 0.000,B 0.000,C 90.000,E1 32.832} C_DIS
LIN {X -0.146,Y -568.292,Z 1504.982,A 0.000,B 0.000,C 90.000,E1 32.801} C_DIS
LIN {X 0.207,Y -395.144,Z 1504.982,A 0.000,B 0.000,C 90.000,E1 32.752} C_DIS
LIN {X -0.199,Y -393.991,Z 1504.978,A 0.000,B 0.000,C 90.000,E1 32.005} C_DIS
LIN {X 0.070,Y -392.684,Z 1504.974,A 0.000,B 0.000,C 90.000,E1 31.258} C_DIS
LIN {X 0.112,Y -385.080,Z 1504.948,A 0.000,B 0.000,C 90.000,E1 26.616} C_DIS
LIN {X 0.079,Y -382.890,Z 1504.938,A 0.000,B 0.000,C 90.000,E1 24.823} C_DIS
LIN {X 0.026,Y -376.182,Z 1504.912,A 0.000,B 0.000,C 90.000,E1 20.120} C_DIS
LIN {X -0.106,Y -373.693,Z 1504.898,A 0.000,B 0.000,C 90.000,E1 17.583} C_DIS
LIN {X 0.030,Y -368.089,Z 1504.869,A 0.000,B 0.000,C 90.000,E1 12.411} C_DIS
LIN {X -0.163,Y -366.410,Z 1504.855,A 0.000,B 0.000,C 90.000,E1 9.849} C_DIS
LIN {X 0.136,Y -361.744,Z 1504.822,A 0.000,B 0.000,C 90.000,E1 3.841} C_DIS
LIN {X 0.022,Y -360.866,Z 1504.801,A 0.000,B 0.000,C 90.000,E1 0.115} C_DIS
LIN {X -0.053,Y -359.426,Z 1504.770,A 0.000,B 0.000,C 90.000,E1 354.546} C_DIS
LIN {X 0.070,Y -358.890,Z 1504.759,A 0.000,B 0.000,C 90.000,E1 352.648} C_DIS
LIN {X -0.020,Y -359.563,Z 1504.726,A 0.000,B 0.000,C 90.000,E1 346.645} C_DIS
LIN {X 0.001,Y -361.801,Z 1504.684,A 0.000,B 0.000,C 90.000,E1 339.135} C_DIS
LIN {X -0.154,Y -362.053,Z 1504.680,A 0.000,B 0.000,C 90.000,E1 338.411} C_DIS
LIN {X 0.189,Y -365.980,Z 1504.643,A 0.000,B 0.000,C 90.000,E1 331.641} C_DIS
LIN {X 0.029,Y -366.387,Z 1504.639,A 0.000,B 0.000,C 90.000,E1 330.923} C_DIS
LIN {X -0.031,Y -371.355,Z 1504.604,A 0.000,B 0.000,C 90.000,E1 324.642} C_DIS
LIN {X -0.043,Y -371.766,Z 1504.602,A 0.000,B 0.000,C 90.000,E1 324.276} C_DIS
LIN {X 0.013,Y -377.358,Z 1504.567,A 0.000,B 0.000,C 90.000,E1 318.038} C_DIS
LIN {X 0.012,Y -378.235,Z 1504.563,A 0.000,B 0.000,C 90.000,E1 317.310} C_DIS
LIN {X 0.002,Y -383.940,Z 1504.531,A 0.000,B 0.000,C 90.000,E1 311.515} C_DIS
LIN {X 0.088,Y -384.893,Z 1504.527,A 0.000,B 0.000,C 90.000,E1 310.782} C_DIS
LIN {X 0.262,Y -390.610,Z 1504.495,A 0.000,B 0.000,C 90.000,E1 305.025} C_DIS
LIN {X 0.106,Y -391.104,Z 1504.493,A 0.000,B 0.000,C 90.000,E1 304.692} C_DIS
LIN {X 0.022,Y -391.648,Z 1504.489,A 0.000,B 0.000,C 90.000,E1 303.992} C_DIS
LIN {X -0.080,Y -396.825,Z 1504.459,A 0.000,B 0.000,C 90.000,E1 298.693} C_DIS
LIN {X -0.210,Y -397.120,Z 1504.457,A 0.000,B 0.000,C 90.000,E1 298.359} C_DIS
LIN {X -0.055,Y -401.597,Z 1504.426,A 0.000,B 0.000,C 90.000,E1 292.717} C_DIS
LIN {X 0.222,Y -404.659,Z 1504.395,A 0.000,B 0.000,C 90.000,E1 287.094} C_DIS
LIN {X -0.079,Y -404.735,Z 1504.391,A 0.000,B 0.000,C 90.000,E1 286.441} C_DIS
LIN {X 0.214,Y -406.099,Z 1504.364,A 0.000,B 0.000,C 90.000,E1 281.535} C_DIS
LIN {X -0.176,Y -406.094,Z 1504.362,A 0.000,B 0.000,C 90.000,E1 281.243} C_DIS
LIN {X -0.097,Y -405.680,Z 1504.333,A 0.000,B 0.000,C 90.000,E1 276.024} C_DIS
LIN {X -0.165,Y -405.058,Z 1504.328,A 0.000,B 0.000,C 90.000,E1 274.992} C_DIS
LIN {X -0.060,Y -403.497,Z 1504.304,A 0.000,B 0.000,C 90.000,E1 270.802} C_DIS
LIN {X -0.092,Y -403.288,Z 1504.302,A 0.000,B 0.000,C 90.000,E1 270.458} C_DIS
LIN {X 0.091,Y -398.931,Z 1504.271,A 0.000,B 0.000,C 90.000,E1 264.837} C_DIS
LIN {X -0.040,Y -393.108,Z 1504.242,A 0.000,B 0.000,C 90.000,E1 259.567} C_DIS
LIN {X -0.079,Y -392.835,Z 1504.240,A 0.000,B 0.000,C 90.000,E1 259.218} C_DIS
LIN {X 0.034,Y -385.993,Z 1504.212,A 0.000,B 0.000,C 90.000,E1 254.212} C_DIS
LIN {X -0.026,Y -385.267,Z 1504.208,A 0.000,B 0.000,C 90.000,E1 253.504} C_DIS
LIN {X -0.004,Y -384.768,Z 1504.206,A 0.000,B 0.000,C 90.000,E1 253.142} C_DIS
LIN {X 0.221,Y -377.973,Z 1504.182,A 0.000,B 0.000,C 90.000,E1 248.773} C_DIS
LIN {X -0.044,Y -376.233,Z 1504.174,A 0.000,B 0.000,C 90.000,E1 247.358} C_DIS
LIN {X 0.057,Y -374.944,Z 1504.170,A 0.000,B 0.000,C 90.000,E1 246.613} C_DIS
LIN {X -0.208,Y -368.417,Z 1504.148,A 0.000,B 0.000,C 90.000,E1 242.615} C_DIS
LIN {X 0.097,Y -366.047,Z 1504.137,A 0.000,B 0.000,C 90.000,E1 240.717} C_DIS
LIN {X 0.004,Y -359.196,Z 1504.115,A 0.000,B 0.000,C 90.000,E1 236.628} C_DIS
LIN {X 0.021,Y -355.842,Z 1504.100,A 0.000,B 0.000,C 90.000,E1 233.989} C_DIS
LIN {X -0.173,Y -348.793,Z 1504.075,A 0.000,B 0.000,C 90.000,E1 229.461} C_DIS
LIN {X -0.097,Y -346.185,Z 1504.062,A 0.000,B 0.000,C 90.000,E1 227.148} C_DIS
LIN {X -0.088,Y -345.065,Z 1504.058,A 0.000,B 0.000,C 90.000,E1 226.377} C_DIS
LIN {X 0.094,Y -338.586,Z 1504.030,A 0.000,B 0.000,C 90.000,E1 221.310} C_DIS
LIN {X 0.094,Y -336.840,Z 1504.019,A 0.000,B 0.000,C 90.000,E1 219.358} C_DIS
LIN {X 0.014,Y -330.861,Z 1503.988,A 0.000,B 0.000,C 90.000,E1 213.865} C_DIS
LIN {X 0.149,Y -329.296,Z 1503.975,A 0.000,B 0.000,C 90.000,E1 211.465} C_DIS
LIN {X -0.154,Y -324.669,Z 1503.942,A 0.000,B 0.000,C 90.000,E1 205.540} C_DIS
LIN {X 0.174,Y -323.837,Z 1503.928,A 0.000,B 0.000,C 90.000,E1 203.078} C_DIS
LIN {X -0.017,Y -321.124,Z 1503.881,A 0.000,B 0.000,C 90.000,E1 194.662} C_DIS
LIN {X 0.138,Y -320.932,Z 1503.877,A 0.000,B 0.000,C 90.000,E1 193.828} C_DIS
LIN {X -0.076,Y -321.562,Z 1503.832,A 0.000,B 0.000,C 90.000,E1 185.796} C_DIS
LIN {X -0.143,Y -324.415,Z 1503.790,A 0.000,B 0.000,C 90.000,E1 178.165} C_DIS
LIN {X -0.141,Y -325.376,Z 1503.783,A 0.000,B 0.000,C 90.000,E1 176.963} C_DIS
LIN {X -0.100,Y -329.112,Z 1503.750,A 0.000,B 0.000,C 90.000,E1 170.971} C_DIS
LIN {X 0.061,Y -334.260,Z 1503.726,A 0.000,B 0.000,C 90.000,E1 166.589} C_DIS
LIN {X 0.067,Y -335.488,Z 1503.719,A 0.000,B 0.000,C 90.000,E1 165.408} C_DIS
LIN {X 0.143,Y -340.932,Z 1503.695,A 0.000,B 0.000,C 90.000,E1 161.094} C_DIS
LIN {X -0.172,Y -342.138,Z 1503.691,A 0.000,B 0.000,C 90.000,E1 160.369} C_DIS
LIN {X -0.058,Y -347.939,Z 1503.667,A 0.000,B 0.000,C 90.000,E1 156.102} C_DIS
LIN {X -0.081,Y -354.259,Z 1503.648,A 0.000,B 0.000,C 90.000,E1 152.666} C_DIS
LIN {X -0.222,Y -361.406,Z 1503.625,A 0.000,B 0.000,C 90.000,E1 148.535} C_DIS
LIN {X 0.137,Y -368.796,Z 1503.606,A 0.000,B 0.000,C 90.000,E1 145.102} C_DIS
LIN {X 0.149,Y -529.931,Z 1503.606,A 0.000,B 0.000,C 90.000,E1 145.102} C_DIS
LIN {X 0.008,Y -530.545,Z 1503.606,A 0.000,B 0.000,C 90.000,E1 145.102} C_DIS
LIN {X -0.339,Y -532.961,Z 1503.605,A 0.000,B 0.000,C 90.000,E1 144.975} C_DIS
LIN {X 0.056,Y -534.395,Z 1503.604,A 0.000,B 0.000,C 90.000,E1 144.769} C_DIS
LIN {X 0.048,Y -536.242,Z 1503.603,A 0.000,B 0.000,C 90.000,E1 144.482} C_DIS
LIN {X -0.103,Y -538.393,Z 1503.600,A 0.000,B 0.000,C 90.000,E1 144.069} C_DIS
LIN {X 0.073,Y -540.077,Z 1503.598,A 0.000,B 0.000,C 90.000,E1 143.623} C_DIS
LIN {X 0.110,Y -541.906,Z 1503.595,A 0.000,B 0.000,C 90.000,E1 143.050} C_DIS
LIN {X 0.162,Y -543.347,Z 1503.592,A 0.000,B 0.000,C 90.000,E1 142.477} C_DIS
LIN {X 0.255,Y -545.065,Z 1503.587,A 0.000,B 0.000,C 90.000,E1 141.618} C_DIS
LIN {X -0.061,Y -546.610,Z 1503.582,A 0.000,B 0.000,C 90.000,E1 140.803} C_DIS
LIN {X 0.079,Y -548.884,Z 1503.574,A 0.000,B 0.000,C 90.000,E1 139.380} C_DIS
LIN {X 0.162,Y -550.162,Z 1503.570,A 0.000,B 0.000,C 90.000,E1 138.528} C_DIS
LIN {X 0.310,Y -551.693,Z 1503.563,A 0.000,B 0.000,C 90.000,E1 137.391} C_DIS
LIN {X 0.068,Y -553.043,Z 1503.557,A 0.000,B 0.000,C 90.000,E1 136.296} C_DIS
LIN {X -0.121,Y -554.600,Z 1503.550,A 0.000,B 0.000,C 90.000,E1 134.919} C_DIS
LIN {X -0.284,Y -555.844,Z 1503.542,A 0.000,B 0.000,C 90.000,E1 133.542} C_DIS
LIN {X -0.060,Y -556.792,Z 1503.536,A 0.000,B 0.000,C 90.000,E1 132.405} C_DIS
LIN {X 0.211,Y -557.714,Z 1503.528,A 0.000,B 0.000,C 90.000,E1 130.987} C_DIS
LIN {X -0.155,Y -558.719,Z 1503.519,A 0.000,B 0.000,C 90.000,E1 129.358} C_DIS
LIN {X 0.033,Y -559.616,Z 1503.508,A 0.000,B 0.000,C 90.000,E1 127.397} C_DIS
LIN {X -0.043,Y -560.080,Z 1503.502,A 0.000,B 0.000,C 90.000,E1 126.297} C_DIS
LIN {X 0.002,Y -560.273,Z 1503.495,A 0.000,B 0.000,C 90.000,E1 125.185} C_DIS
LIN {X 0.057,Y -560.366,Z 1503.489,A 0.000,B 0.000,C 90.000,E1 124.072} C_DIS
LIN {X 0.195,Y -560.220,Z 1503.482,A 0.000,B 0.000,C 90.000,E1 122.673} C_DIS
LIN {X -0.054,Y -560.366,Z 1503.468,A 0.000,B 0.000,C 90.000,E1 120.207} C_DIS
LIN {X -0.236,Y -560.621,Z 1503.459,A 0.000,B 0.000,C 90.000,E1 118.565} C_DIS
LIN {X 0.076,Y -560.901,Z 1503.449,A 0.000,B 0.000,C 90.000,E1 116.873} C_DIS
LIN {X 0.333,Y -561.137,Z 1503.442,A 0.000,B 0.000,C 90.000,E1 115.463} C_DIS
LIN {X 0.040,Y -561.408,Z 1503.436,A 0.000,B 0.000,C 90.000,E1 114.387} C_DIS
LIN {X -0.162,Y -561.724,Z 1503.428,A 0.000,B 0.000,C 90.000,E1 113.025} C_DIS
LIN {X -0.238,Y -562.133,Z 1503.417,A 0.000,B 0.000,C 90.000,E1 111.099} C_DIS
LIN {X 0.221,Y -562.463,Z 1503.408,A 0.000,B 0.000,C 90.000,E1 109.396} C_DIS
LIN {X -0.025,Y -562.829,Z 1503.399,A 0.000,B 0.000,C 90.000,E1 107.764} C_DIS
LIN {X -0.123,Y -563.281,Z 1503.388,A 0.000,B 0.000,C 90.000,E1 105.843} C_DIS
LIN {X -0.288,Y -563.709,Z 1503.380,A 0.000,B 0.000,C 90.000,E1 104.481} C_DIS
LIN {X -0.120,Y -564.280,Z 1503.370,A 0.000,B 0.000,C 90.000,E1 102.535} C_DIS
LIN {X -0.232,Y -564.869,Z 1503.360,A 0.000,B 0.000,C 90.000,E1 100.894} C_DIS
LIN {X 0.117,Y -565.596,Z 1503.351,A 0.000,B 0.000,C 90.000,E1 99.208} C_DIS
LIN {X 0.307,Y -566.167,Z 1503.344,A 0.000,B 0.000,C 90.000,E1 97.814} C_DIS
LIN {X -0.036,Y -566.933,Z 1503.334,A 0.000,B 0.000,C 90.000,E1 96.201} C_DIS
LIN {X -0.095,Y -568.182,Z 1503.322,A 0.000,B 0.000,C 90.000,E1 94.012} C_DIS
LIN {X -0.036,Y -568.919,Z 1503.315,A 0.000,B 0.000,C 90.000,E1 92.636} C_DIS
LIN {X 0.040,Y -569.786,Z 1503.307,A 0.000,B 0.000,C 90.000,E1 91.260} C_DIS
LIN {X -0.055,Y -571.129,Z 1503.295,A 0.000,B 0.000,C 90.000,E1 89.083} C_DIS
LIN {X 0.196,Y -572.124,Z 1503.286,A 0.000,B 0.000,C 90.000,E1 87.421} C_DIS
LIN {X -0.245,Y -572.951,Z 1503.278,A 0.000,B 0.000,C 90.000,E1 86.102} C_DIS
LIN {X 0.253,Y -574.211,Z 1503.268,A 0.000,B 0.000,C 90.000,E1 84.147} C_DIS
LIN {X 0.273,Y -575.476,Z 1503.257,A 0.000,B 0.000,C 90.000,E1 82.243} C_DIS
LIN {X -0.132,Y -576.260,Z 1503.251,A 0.000,B 0.000,C 90.000,E1 81.197} C_DIS
LIN {X 0.014,Y -577.680,Z 1503.240,A 0.000,B 0.000,C 90.000,E1 79.285} C_DIS
LIN {X 0.184,Y -578.957,Z 1503.232,A 0.000,B 0.000,C 90.000,E1 77.645} C_DIS
LIN {X -0.048,Y -580.179,Z 1503.223,A 0.000,B 0.000,C 90.000,E1 76.047} C_DIS
LIN {X 0.315,Y -581.324,Z 1503.214,A 0.000,B 0.000,C 90.000,E1 74.393} C_DIS
LIN {X 0.242,Y -582.027,Z 1503.208,A 0.000,B 0.000,C 90.000,E1 73.323} C_DIS
LIN {X 0.010,Y -582.788,Z 1503.200,A 0.000,B 0.000,C 90.000,E1 72.000} C_DIS
LIN {X -0.300,Y -584.062,Z 1503.188,A 0.000,B 0.000,C 90.000,E1 69.880} C_DIS
LIN {X -0.036,Y -585.057,Z 1503.178,A 0.000,B 0.000,C 90.000,E1 67.975} C_DIS
LIN {X -0.064,Y -586.110,Z 1503.167,A 0.000,B 0.000,C 90.000,E1 66.102} C_DIS
LIN {X 0.064,Y -587.475,Z 1503.155,A 0.000,B 0.000,C 90.000,E1 63.948} C_DIS
LIN {X 0.027,Y -588.388,Z 1503.148,A 0.000,B 0.000,C 90.000,E1 62.615} C_DIS
LIN {X -0.141,Y -589.217,Z 1503.142,A 0.000,B 0.000,C 90.000,E1 61.563} C_DIS
LIN {X 0.000,Y -590.318,Z 1503.133,A 0.000,B 0.000,C 90.000,E1 59.950} C_DIS
LIN {X 0.044,Y -591.272,Z 1503.126,A 0.000,B 0.000,C 90.000,E1 58.614} C_DIS
LIN {X -0.078,Y -592.269,Z 1503.118,A 0.000,B 0.000,C 90.000,E1 57.296} C_DIS
LIN {X 0.113,Y -593.185,Z 1503.112,A 0.000,B 0.000,C 90.000,E1 56.215} C_DIS
LIN {X 0.035,Y -594.120,Z 1503.105,A 0.000,B 0.000,C 90.000,E1 54.895} C_DIS
LIN {X -0.036,Y -594.823,Z 1503.098,A 0.000,B 0.000,C 90.000,E1 53.577} C_DIS
LIN {X -0.224,Y -595.441,Z 1503.090,A 0.000,B 0.000,C 90.000,E1 52.271} C_DIS
LIN {X -0.030,Y -596.281,Z 1503.080,A 0.000,B 0.000,C 90.000,E1 50.400} C_DIS
LIN {X -0.192,Y -596.732,Z 1503.076,A 0.000,B 0.000,C 90.000,E1 49.622} C_DIS
LIN {X 0.195,Y -597.129,Z 1503.070,A 0.000,B 0.000,C 90.000,E1 48.528} C_DIS
LIN {X 0.194,Y -597.164,Z 1503.064,A 0.000,B 0.000,C 90.000,E1 47.472} C_DIS
LIN {X 0.371,Y -597.067,Z 1503.057,A 0.000,B 0.000,C 90.000,E1 46.134} C_DIS
LIN {X -0.083,Y -596.927,Z 1503.051,A 0.000,B 0.000,C 90.000,E1 45.121} C_DIS
LIN {X -0.141,Y -596.076,Z 1503.042,A 0.000,B 0.000,C 90.000,E1 43.542} C_DIS
LIN {X 0.010,Y -595.017,Z 1503.035,A 0.000,B 0.000,C 90.000,E1 42.204} C_DIS
LIN {X -0.023,Y -593.991,Z 1503.029,A 0.000,B 0.000,C 90.000,E1 41.148} C_DIS
LIN {X 0.115,Y -591.740,Z 1503.018,A 0.000,B 0.000,C 90.000,E1 39.277} C_DIS
LIN {X -0.127,Y -589.601,Z 1503.011,A 0.000,B 0.000,C 90.000,E1 37.971} C_DIS
LIN {X -0.182,Y -588.544,Z 1503.008,A 0.000,B 0.000,C 90.000,E1 37.443} C_DIS
LIN {X -0.207,Y -586.275,Z 1503.002,A 0.000,B 0.000,C 90.000,E1 36.377} C_DIS
LIN {X -0.080,Y -582.874,Z 1502.995,A 0.000,B 0.000,C 90.000,E1 35.025} C_DIS
LIN {X -0.056,Y -581.362,Z 1502.992,A 0.000,B 0.000,C 90.000,E1 34.485} C_DIS
LIN {X 0.286,Y -579.520,Z 1502.989,A 0.000,B 0.000,C 90.000,E1 33.913} C_DIS
LIN {X -0.272,Y -576.565,Z 1502.985,A 0.000,B 0.000,C 90.000,E1 33.293} C_DIS
LIN {X -0.120,Y -575.131,Z 1502.983,A 0.000,B 0.000,C 90.000,E1 33.007} C_DIS
LIN {X -0.287,Y -573.360,Z 1502.982,A 0.000,B 0.000,C 90.000,E1 32.752} C_DIS
LIN {X -0.148,Y -571.197,Z 1502.980,A 0.000,B 0.000,C 90.000,E1 32.467} C_DIS
LIN {X 0.004,Y -569.035,Z 1502.979,A 0.000,B 0.000,C 90.000,E1 32.260} C_DIS
LIN {X 0.062,Y -567.400,Z 1502.979,A 0.000,B 0.000,C 90.000,E1 32.163} C_DIS
LIN {X 0.091,Y -566.303,Z 1502.979,A 0.000,B 0.000,C 90.000,E1 32.133} C_DIS
LIN {X 0.039,Y -394.216,Z 1502.979,A 0.000,B 0.000,C 90.000,E1 32.133} C_DIS
LIN {X -0.076,Y -393.560,Z 1502.976,A 0.000,B 0.000,C 90.000,E1 31.720} C_DIS
LIN {X 0.010,Y -386.194,Z 1502.953,A 0.000,B 0.000,C 90.000,E1 27.436} C_DIS
LIN {X 0.158,Y -382.988,Z 1502.938,A 0.000,B 0.000,C 90.000,E1 24.899} C_DIS
LIN {X 0.048,Y -379.071,Z 1502.924,A 0.000,B 0.000,C 90.000,E1 22.386} C_DIS
LIN {X 0.120,Y -373.765,Z 1502.898,A 0.000,B 0.000,C 90.000,E1 17.638} C_DIS
LIN {X 0.067,Y -372.871,Z 1502.894,A 0.000,B 0.000,C 90.000,E1 16.913} C_DIS
LIN {X -0.030,Y -367.601,Z 1502.865,A 0.000,B 0.000,C 90.000,E1 11.771} C_DIS
LIN {X 0.054,Y -366.481,Z 1502.855,A 0.000,B 0.000,C 90.000,E1 9.905} C_DIS
LIN {X -0.010,Y -361.784,Z 1502.822,A 0.000,B 0.000,C 90.000,E1 3.955} C_DIS
LIN {X -0.124,Y -360.899,Z 1502.801,A 0.000,B 0.000,C 90.000,E1 0.229} C_DIS
LIN {X -0.053,Y -359.426,Z 1502.770,A 0.000,B 0.000,C 90.000,E1 354.546} C_DIS
LIN {X 0.070,Y -358.890,Z 1502.759,A 0.000,B 0.000,C 90.000,E1 352.648} C_DIS
LIN {X -0.020,Y -359.563,Z 1502.726,A 0.000,B 0.000,C 90.000,E1 346.645} C_DIS
LIN {X 0.001,Y -361.801,Z 1502.684,A 0.000,B 0.000,C 90.000,E1 339.135} C_DIS
LIN {X -0.154,Y -362.053,Z 1502.680,A 0.000,B 0.000,C 90.000,E1 338.411} C_DIS
LIN {X 0.189,Y -365.980,Z 1502.643,A 0.000,B 0.000,C 90.000,E1 331.641} C_DIS
LIN {X 0.029,Y -366.387,Z 1502.639,A 0.000,B 0.000,C 90.000,E1 330.923} C_DIS
LIN {X -0.031,Y -371.355,Z 1502.604,A 0.000,B 0.000,C 90.000,E1 324.642} C_DIS
LIN {X -0.043,Y -371.766,Z 1502.602,A 0.000,B 0.000,C 90.000,E1 324.276} C_DIS
LIN {X 0.013,Y -377.358,Z 1502.567,A 0.000,B 0.000,C 90.000,E1 318.038} C_DIS
LIN {X 0.012,Y -378.235,Z 1502.563,A 0.000,B 0.000,C 90.000,E1 317.310} C_DIS
LIN {X 0.002,Y -383.940,Z 1502.531,A 0.000,B 0.000,C 90.000,E1 311.515} C_DIS
LIN {X 0.088,Y -384.893,Z 1502.527,A 0.000,B 0.000,C 90.000,E1 310.782} C_DIS
LIN {X 0.262,Y -390.610,Z 1502.495,A 0.000,B 0.000,C 90.000,E1 305.025} C_DIS
LIN {X 0.106,Y -391.104,Z 1502.493,A 0.000,B 0.000,C 90.000,E1 304.692} C_DIS
LIN {X 0.022,Y -391.648,Z 1502.489,A 0.000,B 0.000,C 90.000,E1 303.992} C_DIS
LIN {X -0.080,Y -396.825,Z 1502.459,A 0.000,B 0.000,C 90.000,E1 298.693} C_DIS
LIN {X -0.210,Y -397.120,Z 1502.457,A 0.000,B 0.000,C 90.000,E1 298.359} C_DIS
LIN {X -0.055,Y -401.597,Z 1502.426,A 0.000,B 0.000,C 90.000,E1 292.717} C_DIS
LIN {X 0.222,Y -404.659,Z 1502.395,A 0.000,B 0.000,C 90.000,E1 287.094} C_DIS
LIN {X -0.079,Y -404.735,Z 1502.391,A 0.000,B 0.000,C 90.000,E1 286.441} C_DIS
LIN {X 0.214,Y -406.099,Z 1502.364,A 0.000,B 0.000,C 90.000,E1 281.535} C_DIS
LIN {X -0.176,Y -406.094,Z 1502.362,A 0.000,B 0.000,C 90.000,E1 281.243} C_DIS
LIN {X -0.097,Y -405.680,Z 1502.333,A 0.000,B 0.000,C 90.000,E1 276.024} C_DIS
LIN {X -0.165,Y -405.058,Z 1502.328,A 0.000,B 0.000,C 90.000,E1 274.992} C_DIS
LIN {X -0.060,Y -403.497,Z 1502.304,A 0.000,B 0.000,C 90.000,E1 270.802} C_DIS
LIN {X -0.092,Y -403.288,Z 1502.302,A 0.000,B 0.000,C 90.000,E1 270.458} C_DIS
LIN {X 0.091,Y -398.931,Z 1502.271,A 0.000,B 0.000,C 90.000,E1 264.837} C_DIS
LIN {X -0.040,Y -393.108,Z 1502.242,A 0.000,B 0.000,C 90.000,E1 259.567} C_DIS
LIN {X -0.079,Y -392.835,Z 1502.240,A 0.000,B 0.000,C 90.000,E1 259.218} C_DIS
LIN {X 0.034,Y -385.993,Z 1502.212,A 0.000,B 0.000,C 90.000,E1 254.212} C_DIS
LIN {X -0.026,Y -385.267,Z 1502.208,A 0.000,B 0.000,C 90.000,E1 253.504} C_DIS
LIN {X -0.004,Y -384.768,Z 1502.206,A 0.000,B 0.000,C 90.000,E1 253.142} C_DIS
LIN {X 0.221,Y -377.973,Z 1502.182,A 0.000,B 0.000,C 90.000,E1 248.773} C_DIS
LIN {X -0.044,Y -376.233,Z 1502.174,A 0.000,B 0.000,C 90.000,E1 247.358} C_DIS
LIN {X 0.057,Y -374.944,Z 1502.170,A 0.000,B 0.000,C 90.000,E1 246.613} C_DIS
LIN {X -0.208,Y -368.417,Z 1502.148,A 0.000,B 0.000,C 90.000,E1 242.615} C_DIS
LIN {X 0.097,Y -366.047,Z 1502.137,A 0.000,B 0.000,C 90.000,E1 240.717} C_DIS
LIN {X 0.004,Y -359.196,Z 1502.115,A 0.000,B 0.000,C 90.000,E1 236.628} C_DIS
LIN {X 0.021,Y -355.842,Z 1502.100,A 0.000,B 0.000,C 90.000,E1 233.989} C_DIS
LIN {X -0.173,Y -348.793,Z 1502.075,A 0.000,B 0.000,C 90.000,E1 229.461} C_DIS
LIN {X -0.097,Y -346.185,Z 1502.062,A 0.000,B 0.000,C 90.000,E1 227.148} C_DIS
LIN {X -0.088,Y -345.065,Z 1502.058,A 0.000,B 0.000,C 90.000,E1 226.377} C_DIS
LIN {X 0.094,Y -338.586,Z 1502.030,A 0.000,B 0.000,C 90.000,E1 221.310} C_DIS
LIN {X 0.094,Y -336.840,Z 1502.019,A 0.000,B 0.000,C 90.000,E1 219.358} C_DIS
LIN {X 0.014,Y -330.861,Z 1501.988,A 0.000,B 0.000,C 90.000,E1 213.865} C_DIS
LIN {X 0.149,Y -329.296,Z 1501.975,A 0.000,B 0.000,C 90.000,E1 211.465} C_DIS
LIN {X -0.154,Y -324.669,Z 1501.942,A 0.000,B 0.000,C 90.000,E1 205.540} C_DIS
LIN {X 0.174,Y -323.837,Z 1501.928,A 0.000,B 0.000,C 90.000,E1 203.078} C_DIS
LIN {X -0.017,Y -321.124,Z 1501.881,A 0.000,B 0.000,C 90.000,E1 194.662} C_DIS
LIN {X 0.138,Y -320.932,Z 1501.877,A 0.000,B 0.000,C 90.000,E1 193.828} C_DIS
LIN {X -0.076,Y -321.562,Z 1501.832,A 0.000,B 0.000,C 90.000,E1 185.796} C_DIS
LIN {X -0.143,Y -324.415,Z 1501.790,A 0.000,B 0.000,C 90.000,E1 178.165} C_DIS
LIN {X -0.141,Y -325.376,Z 1501.783,A 0.000,B 0.000,C 90.000,E1 176.963} C_DIS
LIN {X -0.100,Y -329.112,Z 1501.750,A 0.000,B 0.000,C 90.000,E1 170.971} C_DIS
LIN {X 0.061,Y -334.260,Z 1501.726,A 0.000,B 0.000,C 90.000,E1 166.589} C_DIS
LIN {X 0.067,Y -335.488,Z 1501.719,A 0.000,B 0.000,C 90.000,E1 165.408} C_DIS
LIN {X 0.143,Y -340.932,Z 1501.695,A 0.000,B 0.000,C 90.000,E1 161.094} C_DIS
LIN {X -0.172,Y -342.138,Z 1501.691,A 0.000,B 0.000,C 90.000,E1 160.369} C_DIS
LIN {X -0.058,Y -347.939,Z 1501.667,A 0.000,B 0.000,C 90.000,E1 156.102} C_DIS
LIN {X -0.081,Y -354.259,Z 1501.648,A 0.000,B 0.000,C 90.000,E1 152.666} C_DIS
LIN {X -0.222,Y -361.406,Z 1501.625,A 0.000,B 0.000,C 90.000,E1 148.535} C_DIS
LIN {X -0.200,Y -367.126,Z 1501.610,A 0.000,B 0.000,C 90.000,E1 145.881} C_DIS
LIN {X -0.335,Y -528.295,Z 1501.610,A 0.000,B 0.000,C 90.000,E1 145.881} C_DIS
LIN {X 0.052,Y -531.203,Z 1501.609,A 0.000,B 0.000,C 90.000,E1 145.674} C_DIS
LIN {X 0.002,Y -532.710,Z 1501.609,A 0.000,B 0.000,C 90.000,E1 145.515} C_DIS
LIN {X 0.035,Y -534.635,Z 1501.607,A 0.000,B 0.000,C 90.000,E1 145.229} C_DIS
LIN {X -0.120,Y -536.925,Z 1501.604,A 0.000,B 0.000,C 90.000,E1 144.815} C_DIS
LIN {X -0.267,Y -538.684,Z 1501.602,A 0.000,B 0.000,C 90.000,E1 144.402} C_DIS
LIN {X 0.180,Y -539.713,Z 1501.601,A 0.000,B 0.000,C 90.000,E1 144.069} C_DIS
LIN {X 0.212,Y -541.407,Z 1501.597,A 0.000,B 0.000,C 90.000,E1 143.497} C_DIS
LIN {X -0.147,Y -543.404,Z 1501.593,A 0.000,B 0.000,C 90.000,E1 142.683} C_DIS
LIN {X -0.051,Y -545.163,Z 1501.588,A 0.000,B 0.000,C 90.000,E1 141.823} C_DIS
LIN {X 0.060,Y -546.706,Z 1501.583,A 0.000,B 0.000,C 90.000,E1 140.964} C_DIS
LIN {X 0.154,Y -548.548,Z 1501.577,A 0.000,B 0.000,C 90.000,E1 139.828} C_DIS
LIN {X 0.281,Y -550.263,Z 1501.571,A 0.000,B 0.000,C 90.000,E1 138.690} C_DIS
LIN {X 0.021,Y -551.792,Z 1501.564,A 0.000,B 0.000,C 90.000,E1 137.595} C_DIS
LIN {X 0.188,Y -553.157,Z 1501.558,A 0.000,B 0.000,C 90.000,E1 136.458} C_DIS
LIN {X 0.001,Y -554.717,Z 1501.551,A 0.000,B 0.000,C 90.000,E1 135.081} C_DIS
LIN {X -0.160,Y -555.969,Z 1501.543,A 0.000,B 0.000,C 90.000,E1 133.704} C_DIS
LIN {X 0.099,Y -557.102,Z 1501.535,A 0.000,B 0.000,C 90.000,E1 132.285} C_DIS
LIN {X -0.001,Y -558.005,Z 1501.527,A 0.000,B 0.000,C 90.000,E1 130.906} C_DIS
LIN {X -0.017,Y -558.839,Z 1501.520,A 0.000,B 0.000,C 90.000,E1 129.519} C_DIS
LIN {X 0.340,Y -559.434,Z 1501.512,A 0.000,B 0.000,C 90.000,E1 128.096} C_DIS
LIN {X -0.078,Y -559.968,Z 1501.506,A 0.000,B 0.000,C 90.000,E1 127.030} C_DIS
LIN {X -0.157,Y -560.247,Z 1501.500,A 0.000,B 0.000,C 90.000,E1 125.931} C_DIS
LIN {X -0.111,Y -560.399,Z 1501.493,A 0.000,B 0.000,C 90.000,E1 124.818} C_DIS
LIN {X -0.060,Y -560.394,Z 1501.487,A 0.000,B 0.000,C 90.000,E1 123.706} C_DIS
LIN {X -0.141,Y -560.343,Z 1501.470,A 0.000,B 0.000,C 90.000,E1 120.669} C_DIS
LIN {X -0.052,Y -560.588,Z 1501.461,A 0.000,B 0.000,C 90.000,E1 118.999} C_DIS
LIN {X -0.007,Y -560.871,Z 1501.452,A 0.000,B 0.000,C 90.000,E1 117.334} C_DIS
LIN {X 0.057,Y -561.140,Z 1501.443,A 0.000,B 0.000,C 90.000,E1 115.668} C_DIS
LIN {X 0.082,Y -561.456,Z 1501.435,A 0.000,B 0.000,C 90.000,E1 114.283} C_DIS
LIN {X 0.112,Y -561.785,Z 1501.427,A 0.000,B 0.000,C 90.000,E1 112.898} C_DIS
LIN {X 0.240,Y -562.136,Z 1501.418,A 0.000,B 0.000,C 90.000,E1 111.227} C_DIS
LIN {X 0.173,Y -562.505,Z 1501.409,A 0.000,B 0.000,C 90.000,E1 109.577} C_DIS
LIN {X 0.241,Y -562.917,Z 1501.398,A 0.000,B 0.000,C 90.000,E1 107.638} C_DIS
LIN {X 0.138,Y -563.377,Z 1501.387,A 0.000,B 0.000,C 90.000,E1 105.717} C_DIS
LIN {X -0.030,Y -563.797,Z 1501.380,A 0.000,B 0.000,C 90.000,E1 104.356} C_DIS
LIN {X 0.130,Y -564.396,Z 1501.369,A 0.000,B 0.000,C 90.000,E1 102.411} C_DIS
LIN {X -0.094,Y -565.009,Z 1501.360,A 0.000,B 0.000,C 90.000,E1 100.782} C_DIS
LIN {X -0.295,Y -565.737,Z 1501.351,A 0.000,B 0.000,C 90.000,E1 99.151} C_DIS
LIN {X -0.101,Y -566.307,Z 1501.343,A 0.000,B 0.000,C 90.000,E1 97.757} C_DIS
LIN {X 0.287,Y -567.213,Z 1501.332,A 0.000,B 0.000,C 90.000,E1 95.796} C_DIS
LIN {X -0.082,Y -568.180,Z 1501.323,A 0.000,B 0.000,C 90.000,E1 94.188} C_DIS
LIN {X -0.105,Y -568.828,Z 1501.317,A 0.000,B 0.000,C 90.000,E1 93.094} C_DIS
LIN {X 0.219,Y -569.971,Z 1501.307,A 0.000,B 0.000,C 90.000,E1 91.146} C_DIS
LIN {X -0.003,Y -571.180,Z 1501.296,A 0.000,B 0.000,C 90.000,E1 89.255} C_DIS
LIN {X 0.252,Y -572.252,Z 1501.287,A 0.000,B 0.000,C 90.000,E1 87.593} C_DIS
LIN {X -0.050,Y -573.239,Z 1501.278,A 0.000,B 0.000,C 90.000,E1 85.988} C_DIS
LIN {X -0.120,Y -574.511,Z 1501.267,A 0.000,B 0.000,C 90.000,E1 84.090} C_DIS
LIN {X 0.108,Y -576.008,Z 1501.255,A 0.000,B 0.000,C 90.000,E1 81.894} C_DIS
LIN {X 0.282,Y -576.778,Z 1501.249,A 0.000,B 0.000,C 90.000,E1 80.792} C_DIS
LIN {X -0.239,Y -578.036,Z 1501.240,A 0.000,B 0.000,C 90.000,E1 79.218} C_DIS
LIN {X 0.045,Y -579.519,Z 1501.229,A 0.000,B 0.000,C 90.000,E1 77.297} C_DIS
LIN {X -0.179,Y -580.713,Z 1501.220,A 0.000,B 0.000,C 90.000,E1 75.700} C_DIS
LIN {X -0.037,Y -581.679,Z 1501.213,A 0.000,B 0.000,C 90.000,E1 74.338} C_DIS
LIN {X 0.279,Y -582.504,Z 1501.206,A 0.000,B 0.000,C 90.000,E1 72.960} C_DIS
LIN {X 0.057,Y -583.262,Z 1501.198,A 0.000,B 0.000,C 90.000,E1 71.638} C_DIS
LIN {X 0.102,Y -584.368,Z 1501.188,A 0.000,B 0.000,C 90.000,E1 69.752} C_DIS
LIN {X 0.027,Y -585.548,Z 1501.176,A 0.000,B 0.000,C 90.000,E1 67.614} C_DIS
LIN {X 0.002,Y -586.591,Z 1501.165,A 0.000,B 0.000,C 90.000,E1 65.741} C_DIS
LIN {X -0.284,Y -587.810,Z 1501.155,A 0.000,B 0.000,C 90.000,E1 63.896} C_DIS
LIN {X -0.053,Y -588.718,Z 1501.147,A 0.000,B 0.000,C 90.000,E1 62.538} C_DIS
LIN {X 0.026,Y -589.529,Z 1501.141,A 0.000,B 0.000,C 90.000,E1 61.463} C_DIS
LIN {X 0.052,Y -590.476,Z 1501.134,A 0.000,B 0.000,C 90.000,E1 60.127} C_DIS
LIN {X -0.003,Y -591.606,Z 1501.125,A 0.000,B 0.000,C 90.000,E1 58.535} C_DIS
LIN {X 0.062,Y -592.640,Z 1501.118,A 0.000,B 0.000,C 90.000,E1 57.199} C_DIS
LIN {X 0.084,Y -593.531,Z 1501.112,A 0.000,B 0.000,C 90.000,E1 56.135} C_DIS
LIN {X 0.016,Y -594.450,Z 1501.105,A 0.000,B 0.000,C 90.000,E1 54.815} C_DIS
LIN {X -0.270,Y -595.099,Z 1501.099,A 0.000,B 0.000,C 90.000,E1 53.783} C_DIS
LIN {X 0.021,Y -595.690,Z 1501.091,A 0.000,B 0.000,C 90.000,E1 52.431} C_DIS
LIN {X -0.165,Y -596.562,Z 1501.081,A 0.000,B 0.000,C 90.000,E1 50.598} C_DIS
LIN {X -0.176,Y -597.133,Z 1501.075,A 0.000,B 0.000,C 90.000,E1 49.542} C_DIS
LIN {X -0.177,Y -597.477,Z 1501.069,A 0.000,B 0.000,C 90.000,E1 48.485} C_DIS
LIN {X 0.224,Y -597.533,Z 1501.063,A 0.000,B 0.000,C 90.000,E1 47.391} C_DIS
LIN {X -0.218,Y -597.468,Z 1501.058,A 0.000,B 0.000,C 90.000,E1 46.377} C_DIS
LIN {X -0.042,Y -597.242,Z 1501.050,A 0.000,B 0.000,C 90.000,E1 45.040} C_DIS
LIN {X 0.127,Y -596.534,Z 1501.043,A 0.000,B 0.000,C 90.000,E1 43.704} C_DIS
LIN {X -0.327,Y -595.761,Z 1501.037,A 0.000,B 0.000,C 90.000,E1 42.690} C_DIS
LIN {X 0.263,Y -594.577,Z 1501.030,A 0.000,B 0.000,C 90.000,E1 41.310} C_DIS
LIN {X 0.204,Y -592.649,Z 1501.021,A 0.000,B 0.000,C 90.000,E1 39.725} C_DIS
LIN {X 0.174,Y -591.999,Z 1501.018,A 0.000,B 0.000,C 90.000,E1 39.197} C_DIS
LIN {X -0.065,Y -589.834,Z 1501.010,A 0.000,B 0.000,C 90.000,E1 37.890} C_DIS
LIN {X 0.283,Y -587.695,Z 1501.005,A 0.000,B 0.000,C 90.000,E1 36.790} C_DIS
LIN {X 0.050,Y -585.858,Z 1501.000,A 0.000,B 0.000,C 90.000,E1 36.011} C_DIS
LIN {X -0.017,Y -583.135,Z 1500.994,A 0.000,B 0.000,C 90.000,E1 34.945} C_DIS
LIN {X 0.009,Y -581.609,Z 1500.991,A 0.000,B 0.000,C 90.000,E1 34.405} C_DIS
LIN {X 0.028,Y -579.887,Z 1500.988,A 0.000,B 0.000,C 90.000,E1 33.865} C_DIS
LIN {X 0.356,Y -577.980,Z 1500.985,A 0.000,B 0.000,C 90.000,E1 33.293} C_DIS
LIN {X -0.367,Y -576.274,Z 1500.983,A 0.000,B 0.000,C 90.000,E1 32.959} C_DIS
LIN {X -0.298,Y -574.187,Z 1500.981,A 0.000,B 0.000,C 90.000,E1 32.546} C_DIS
LIN {X -0.244,Y -571.536,Z 1500.978,A 0.000,B 0.000,C 90.000,E1 32.133} C_DIS
LIN {X 0.367,Y -569.285,Z 1500.977,A 0.000,B 0.000,C 90.000,E1 31.799} C_DIS
LIN {X -0.269,Y -567.127,Z 1500.976,A 0.000,B 0.000,C 90.000,E1 31.671} C_DIS
LIN {X 0.090,Y -565.603,Z 1500.975,A 0.000,B 0.000,C 90.000,E1 31.544} C_DIS
LIN {X -0.024,Y -564.256,Z 1500.975,A 0.000,B 0.000,C 90.000,E1 31.514} C_DIS
LIN {X -0.059,Y -563.898,Z 1500.975,A 0.000,B 0.000,C 90.000,E1 31.514} C_DIS
LIN {X -0.064,Y -393.149,Z 1500.975,A 0.000,B 0.000,C 90.000,E1 31.514} C_DIS
LIN {X -0.060,Y -385.815,Z 1500.951,A 0.000,B 0.000,C 90.000,E1 27.180} C_DIS
LIN {X -0.080,Y -383.092,Z 1500.939,A 0.000,B 0.000,C 90.000,E1 25.027} C_DIS
LIN {X 0.078,Y -381.999,Z 1500.935,A 0.000,B 0.000,C 90.000,E1 24.283} C_DIS
LIN {X 0.002,Y -375.582,Z 1500.909,A 0.000,B 0.000,C 90.000,E1 19.577} C_DIS
LIN {X -0.118,Y -373.500,Z 1500.897,A 0.000,B 0.000,C 90.000,E1 17.402} C_DIS
LIN {X -0.079,Y -367.945,Z 1500.868,A 0.000,B 0.000,C 90.000,E1 12.243} C_DIS
LIN {X -0.059,Y -366.529,Z 1500.856,A 0.000,B 0.000,C 90.000,E1 10.018} C_DIS
LIN {X 0.084,Y -365.037,Z 1500.847,A 0.000,B 0.000,C 90.000,E1 8.511} C_DIS
LIN {X 0.179,Y -361.084,Z 1500.810,A 0.000,B 0.000,C 90.000,E1 1.776} C_DIS
LIN {X 0.120,Y -360.905,Z 1500.802,A 0.000,B 0.000,C 90.000,E1 0.286} C_DIS
LIN {X -0.053,Y -359.426,Z 1500.770,A 0.000,B 0.000,C 90.000,E1 354.546} C_DIS
LIN {X 0.070,Y -358.890,Z 1500.759,A 0.000,B 0.000,C 90.000,E1 352.648} C_DIS
LIN {X -0.020,Y -359.563,Z 1500.726,A 0.000,B 0.000,C 90.000,E1 346.645} C_DIS
LIN {X 0.001,Y -361.801,Z 1500.684,A 0.000,B 0.000,C 90.000,E1 339.135} C_DIS
LIN {X -0.154,Y -362.053,Z 1500.680,A 0.000,B 0.000,C 90.000,E1 338.411} C_DIS
LIN {X 0.189,Y -365.980,Z 1500.643,A 0.000,B 0.000,C 90.000,E1 331.641} C_DIS
LIN {X 0.029,Y -366.387,Z 1500.639,A 0.000,B 0.000,C 90.000,E1 330.923} C_DIS
LIN {X -0.031,Y -371.355,Z 1500.604,A 0.000,B 0.000,C 90.000,E1 324.642} C_DIS
LIN {X -0.043,Y -371.766,Z 1500.602,A 0.000,B 0.000,C 90.000,E1 324.276} C_DIS
LIN {X 0.013,Y -377.358,Z 1500.567,A 0.000,B 0.000,C 90.000,E1 318.038} C_DIS
LIN {X 0.012,Y -378.235,Z 1500.563,A 0.000,B 0.000,C 90.000,E1 317.310} C_DIS
LIN {X 0.002,Y -383.940,Z 1500.531,A 0.000,B 0.000,C 90.000,E1 311.515} C_DIS
LIN {X 0.088,Y -384.893,Z 1500.527,A 0.000,B 0.000,C 90.000,E1 310.782} C_DIS
LIN {X 0.262,Y -390.610,Z 1500.495,A 0.000,B 0.000,C 90.000,E1 305.025} C_DIS
LIN {X 0.106,Y -391.104,Z 1500.493,A 0.000,B 0.000,C 90.000,E1 304.692} C_DIS
LIN {X 0.022,Y -391.648,Z 1500.489,A 0.000,B 0.000,C 90.000,E1 303.992} C_DIS
LIN {X -0.080,Y -396.825,Z 1500.459,A 0.000,B 0.000,C 90.000,E1 298.693} C_DIS
LIN {X -0.210,Y -397.120,Z 1500.457,A 0.000,B 0.000,C 90.000,E1 298.359} C_DIS
LIN {X -0.055,Y -401.597,Z 1500.426,A 0.000,B 0.000,C 90.000,E1 292.717} C_DIS
LIN {X 0.222,Y -404.659,Z 1500.395,A 0.000,B 0.000,C 90.000,E1 287.094} C_DIS
LIN {X -0.079,Y -404.735,Z 1500.391,A 0.000,B 0.000,C 90.000,E1 286.441} C_DIS
LIN {X 0.214,Y -406.099,Z 1500.364,A 0.000,B 0.000,C 90.000,E1 281.535} C_DIS
LIN {X -0.176,Y -406.094,Z 1500.362,A 0.000,B 0.000,C 90.000,E1 281.243} C_DIS
LIN {X -0.097,Y -405.680,Z 1500.333,A 0.000,B 0.000,C 90.000,E1 276.024} C_DIS
LIN {X -0.165,Y -405.058,Z 1500.328,A 0.000,B 0.000,C 90.000,E1 274.992} C_DIS
LIN {X -0.060,Y -403.497,Z 1500.304,A 0.000,B 0.000,C 90.000,E1 270.802} C_DIS
LIN {X -0.092,Y -403.288,Z 1500.302,A 0.000,B 0.000,C 90.000,E1 270.458} C_DIS
LIN {X 0.091,Y -398.931,Z 1500.271,A 0.000,B 0.000,C 90.000,E1 264.837} C_DIS
LIN {X -0.040,Y -393.108,Z 1500.242,A 0.000,B 0.000,C 90.000,E1 259.567} C_DIS
LIN {X -0.079,Y -392.835,Z 1500.240,A 0.000,B 0.000,C 90.000,E1 259.218} C_DIS
LIN {X 0.034,Y -385.993,Z 1500.212,A 0.000,B 0.000,C 90.000,E1 254.212} C_DIS
LIN {X -0.026,Y -385.267,Z 1500.208,A 0.000,B 0.000,C 90.000,E1 253.504} C_DIS
LIN {X -0.004,Y -384.768,Z 1500.206,A 0.000,B 0.000,C 90.000,E1 253.142} C_DIS
LIN {X 0.221,Y -377.973,Z 1500.182,A 0.000,B 0.000,C 90.000,E1 248.773} C_DIS
LIN {X -0.044,Y -376.233,Z 1500.174,A 0.000,B 0.000,C 90.000,E1 247.358} C_DIS
LIN {X 0.057,Y -374.944,Z 1500.170,A 0.000,B 0.000,C 90.000,E1 246.613} C_DIS
LIN {X -0.208,Y -368.417,Z 1500.148,A 0.000,B 0.000,C 90.000,E1 242.615} C_DIS
LIN {X 0.097,Y -366.047,Z 1500.137,A 0.000,B 0.000,C 90.000,E1 240.717} C_DIS
LIN {X 0.004,Y -359.196,Z 1500.115,A 0.000,B 0.000,C 90.000,E1 236.628} C_DIS
LIN {X 0.021,Y -355.842,Z 1500.100,A 0.000,B 0.000,C 90.000,E1 233.989} C_DIS
LIN {X -0.173,Y -348.793,Z 1500.075,A 0.000,B 0.000,C 90.000,E1 229.461} C_DIS
LIN {X -0.097,Y -346.185,Z 1500.062,A 0.000,B 0.000,C 90.000,E1 227.148} C_DIS
LIN {X -0.088,Y -345.065,Z 1500.058,A 0.000,B 0.000,C 90.000,E1 226.377} C_DIS
LIN {X 0.094,Y -338.586,Z 1500.030,A 0.000,B 0.000,C 90.000,E1 221.310} C_DIS
LIN {X 0.094,Y -336.840,Z 1500.019,A 0.000,B 0.000,C 90.000,E1 219.358} C_DIS
LIN {X 0.014,Y -330.861,Z 1499.988,A 0.000,B 0.000,C 90.000,E1 213.865} C_DIS
LIN {X 0.149,Y -329.296,Z 1499.975,A 0.000,B 0.000,C 90.000,E1 211.465} C_DIS
LIN {X -0.154,Y -324.669,Z 1499.942,A 0.000,B 0.000,C 90.000,E1 205.540} C_DIS
LIN {X 0.174,Y -323.837,Z 1499.928,A 0.000,B 0.000,C 90.000,E1 203.078} C_DIS
LIN {X -0.017,Y -321.124,Z 1499.881,A 0.000,B 0.000,C 90.000,E1 194.662} C_DIS
LIN {X 0.138,Y -320.932,Z 1499.877,A 0.000,B 0.000,C 90.000,E1 193.828} C_DIS
LIN {X -0.076,Y -321.562,Z 1499.832,A 0.000,B 0.000,C 90.000,E1 185.796} C_DIS
LIN {X -0.143,Y -324.415,Z 1499.790,A 0.000,B 0.000,C 90.000,E1 178.165} C_DIS
LIN {X -0.141,Y -325.376,Z 1499.783,A 0.000,B 0.000,C 90.000,E1 176.963} C_DIS
LIN {X -0.100,Y -329.112,Z 1499.750,A 0.000,B 0.000,C 90.000,E1 170.971} C_DIS
LIN {X 0.061,Y -334.260,Z 1499.726,A 0.000,B 0.000,C 90.000,E1 166.589} C_DIS
LIN {X 0.067,Y -335.488,Z 1499.719,A 0.000,B 0.000,C 90.000,E1 165.408} C_DIS
LIN {X 0.143,Y -340.932,Z 1499.695,A 0.000,B 0.000,C 90.000,E1 161.094} C_DIS
LIN {X -0.172,Y -342.138,Z 1499.691,A 0.000,B 0.000,C 90.000,E1 160.369} C_DIS
LIN {X -0.058,Y -347.939,Z 1499.667,A 0.000,B 0.000,C 90.000,E1 156.102} C_DIS
LIN {X -0.081,Y -354.259,Z 1499.648,A 0.000,B 0.000,C 90.000,E1 152.666} C_DIS
LIN {X -0.222,Y -361.406,Z 1499.625,A 0.000,B 0.000,C 90.000,E1 148.535} C_DIS
LIN {X -0.096,Y -365.486,Z 1499.614,A 0.000,B 0.000,C 90.000,E1 146.580} C_DIS
LIN {X 0.109,Y -526.345,Z 1499.614,A 0.000,B 0.000,C 90.000,E1 146.548} C_DIS
LIN {X 0.026,Y -526.893,Z 1499.614,A 0.000,B 0.000,C 90.000,E1 146.548} C_DIS
LIN {X -0.152,Y -529.404,Z 1499.613,A 0.000,B 0.000,C 90.000,E1 146.421} C_DIS
LIN {X -0.330,Y -530.851,Z 1499.613,A 0.000,B 0.000,C 90.000,E1 146.294} C_DIS
LIN {X -0.120,Y -531.941,Z 1499.612,A 0.000,B 0.000,C 90.000,E1 146.135} C_DIS
LIN {X -0.061,Y -533.686,Z 1499.610,A 0.000,B 0.000,C 90.000,E1 145.849} C_DIS
LIN {X 0.218,Y -535.876,Z 1499.608,A 0.000,B 0.000,C 90.000,E1 145.388} C_DIS
LIN {X -0.083,Y -538.200,Z 1499.605,A 0.000,B 0.000,C 90.000,E1 144.848} C_DIS
LIN {X -0.065,Y -540.000,Z 1499.602,A 0.000,B 0.000,C 90.000,E1 144.276} C_DIS
LIN {X -0.008,Y -542.159,Z 1499.597,A 0.000,B 0.000,C 90.000,E1 143.417} C_DIS
LIN {X 0.139,Y -545.246,Z 1499.589,A 0.000,B 0.000,C 90.000,E1 141.984} C_DIS
LIN {X -0.137,Y -547.261,Z 1499.583,A 0.000,B 0.000,C 90.000,E1 140.884} C_DIS
LIN {X -0.034,Y -549.093,Z 1499.576,A 0.000,B 0.000,C 90.000,E1 139.747} C_DIS
LIN {X 0.102,Y -550.744,Z 1499.570,A 0.000,B 0.000,C 90.000,E1 138.609} C_DIS
LIN {X 0.256,Y -552.265,Z 1499.564,A 0.000,B 0.000,C 90.000,E1 137.472} C_DIS
LIN {X -0.330,Y -553.897,Z 1499.556,A 0.000,B 0.000,C 90.000,E1 136.134} C_DIS
LIN {X -0.158,Y -555.101,Z 1499.550,A 0.000,B 0.000,C 90.000,E1 135.000} C_DIS
LIN {X 0.091,Y -556.339,Z 1499.542,A 0.000,B 0.000,C 90.000,E1 133.581} C_DIS
LIN {X -0.048,Y -557.411,Z 1499.535,A 0.000,B 0.000,C 90.000,E1 132.204} C_DIS
LIN {X 0.201,Y -558.131,Z 1499.528,A 0.000,B 0.000,C 90.000,E1 131.067} C_DIS
LIN {X -0.241,Y -558.926,Z 1499.521,A 0.000,B 0.000,C 90.000,E1 129.725} C_DIS
LIN {X 0.113,Y -559.546,Z 1499.513,A 0.000,B 0.000,C 90.000,E1 128.302} C_DIS
LIN {X -0.214,Y -560.110,Z 1499.505,A 0.000,B 0.000,C 90.000,E1 126.950} C_DIS
LIN {X 0.254,Y -560.395,Z 1499.498,A 0.000,B 0.000,C 90.000,E1 125.518} C_DIS
LIN {X 0.306,Y -560.430,Z 1499.491,A 0.000,B 0.000,C 90.000,E1 124.405} C_DIS
LIN {X 0.356,Y -560.353,Z 1499.485,A 0.000,B 0.000,C 90.000,E1 123.293} C_DIS
LIN {X -0.081,Y -560.350,Z 1499.471,A 0.000,B 0.000,C 90.000,E1 120.846} C_DIS
LIN {X 0.013,Y -560.633,Z 1499.461,A 0.000,B 0.000,C 90.000,E1 118.899} C_DIS
LIN {X -0.166,Y -560.899,Z 1499.451,A 0.000,B 0.000,C 90.000,E1 117.257} C_DIS
LIN {X 0.197,Y -561.228,Z 1499.441,A 0.000,B 0.000,C 90.000,E1 115.283} C_DIS
LIN {X 0.223,Y -561.537,Z 1499.433,A 0.000,B 0.000,C 90.000,E1 113.898} C_DIS
LIN {X -0.068,Y -561.842,Z 1499.427,A 0.000,B 0.000,C 90.000,E1 112.823} C_DIS
LIN {X 0.169,Y -562.245,Z 1499.416,A 0.000,B 0.000,C 90.000,E1 110.865} C_DIS
LIN {X 0.108,Y -562.622,Z 1499.407,A 0.000,B 0.000,C 90.000,E1 109.214} C_DIS
LIN {X -0.135,Y -562.996,Z 1499.398,A 0.000,B 0.000,C 90.000,E1 107.583} C_DIS
LIN {X 0.159,Y -563.417,Z 1499.388,A 0.000,B 0.000,C 90.000,E1 105.898} C_DIS
LIN {X 0.153,Y -563.877,Z 1499.379,A 0.000,B 0.000,C 90.000,E1 104.245} C_DIS
LIN {X 0.161,Y -564.414,Z 1499.370,A 0.000,B 0.000,C 90.000,E1 102.591} C_DIS
LIN {X 0.215,Y -565.142,Z 1499.359,A 0.000,B 0.000,C 90.000,E1 100.658} C_DIS
LIN {X 0.007,Y -565.876,Z 1499.350,A 0.000,B 0.000,C 90.000,E1 99.029} C_DIS
LIN {X -0.049,Y -566.340,Z 1499.344,A 0.000,B 0.000,C 90.000,E1 97.936} C_DIS
LIN {X -0.050,Y -567.402,Z 1499.332,A 0.000,B 0.000,C 90.000,E1 95.739} C_DIS
LIN {X 0.153,Y -568.335,Z 1499.323,A 0.000,B 0.000,C 90.000,E1 94.073} C_DIS
LIN {X 0.133,Y -569.003,Z 1499.317,A 0.000,B 0.000,C 90.000,E1 92.980} C_DIS
LIN {X -0.234,Y -570.022,Z 1499.308,A 0.000,B 0.000,C 90.000,E1 91.375} C_DIS
LIN {X 0.248,Y -571.405,Z 1499.295,A 0.000,B 0.000,C 90.000,E1 89.141} C_DIS
LIN {X -0.201,Y -572.340,Z 1499.288,A 0.000,B 0.000,C 90.000,E1 87.822} C_DIS
LIN {X 0.074,Y -573.354,Z 1499.279,A 0.000,B 0.000,C 90.000,E1 86.159} C_DIS
LIN {X 0.013,Y -574.616,Z 1499.268,A 0.000,B 0.000,C 90.000,E1 84.261} C_DIS
LIN {X 0.090,Y -575.334,Z 1499.262,A 0.000,B 0.000,C 90.000,E1 83.166} C_DIS
LIN {X 0.221,Y -576.748,Z 1499.252,A 0.000,B 0.000,C 90.000,E1 81.254} C_DIS
LIN {X -0.184,Y -578.167,Z 1499.241,A 0.000,B 0.000,C 90.000,E1 79.398} C_DIS
LIN {X 0.224,Y -579.661,Z 1499.231,A 0.000,B 0.000,C 90.000,E1 77.465} C_DIS
LIN {X -0.129,Y -580.880,Z 1499.222,A 0.000,B 0.000,C 90.000,E1 75.880} C_DIS
LIN {X -0.167,Y -582.022,Z 1499.213,A 0.000,B 0.000,C 90.000,E1 74.267} C_DIS
LIN {X -0.006,Y -582.835,Z 1499.205,A 0.000,B 0.000,C 90.000,E1 72.906} C_DIS
LIN {X -0.228,Y -583.595,Z 1499.198,A 0.000,B 0.000,C 90.000,E1 71.583} C_DIS
LIN {X -0.181,Y -584.670,Z 1499.187,A 0.000,B 0.000,C 90.000,E1 69.699} C_DIS
LIN {X -0.033,Y -585.895,Z 1499.175,A 0.000,B 0.000,C 90.000,E1 67.539} C_DIS
LIN {X -0.040,Y -586.946,Z 1499.165,A 0.000,B 0.000,C 90.000,E1 65.665} C_DIS
LIN {X 0.219,Y -588.142,Z 1499.154,A 0.000,B 0.000,C 90.000,E1 63.768} C_DIS
LIN {X -0.337,Y -589.045,Z 1499.147,A 0.000,B 0.000,C 90.000,E1 62.487} C_DIS
LIN {X 0.022,Y -589.835,Z 1499.141,A 0.000,B 0.000,C 90.000,E1 61.385} C_DIS
LIN {X -0.048,Y -590.951,Z 1499.132,A 0.000,B 0.000,C 90.000,E1 59.793} C_DIS
LIN {X -0.093,Y -592.126,Z 1499.123,A 0.000,B 0.000,C 90.000,E1 58.201} C_DIS
LIN {X 0.301,Y -593.203,Z 1499.116,A 0.000,B 0.000,C 90.000,E1 56.834} C_DIS
LIN {X 0.007,Y -594.071,Z 1499.110,A 0.000,B 0.000,C 90.000,E1 55.801} C_DIS
LIN {X -0.058,Y -594.985,Z 1499.103,A 0.000,B 0.000,C 90.000,E1 54.482} C_DIS
LIN {X -0.216,Y -595.506,Z 1499.098,A 0.000,B 0.000,C 90.000,E1 53.703} C_DIS
LIN {X 0.085,Y -596.047,Z 1499.091,A 0.000,B 0.000,C 90.000,E1 52.351} C_DIS
LIN {X -0.089,Y -596.959,Z 1499.081,A 0.000,B 0.000,C 90.000,E1 50.517} C_DIS
LIN {X -0.093,Y -597.520,Z 1499.075,A 0.000,B 0.000,C 90.000,E1 49.461} C_DIS
LIN {X -0.088,Y -597.838,Z 1499.069,A 0.000,B 0.000,C 90.000,E1 48.405} C_DIS
LIN {X 0.318,Y -597.904,Z 1499.063,A 0.000,B 0.000,C 90.000,E1 47.310} C_DIS
LIN {X 0.100,Y -597.874,Z 1499.059,A 0.000,B 0.000,C 90.000,E1 46.539} C_DIS
LIN {X -0.141,Y -597.658,Z 1499.051,A 0.000,B 0.000,C 90.000,E1 45.243} C_DIS
LIN {X -0.384,Y -596.994,Z 1499.044,A 0.000,B 0.000,C 90.000,E1 43.947} C_DIS
LIN {X 0.233,Y -596.479,Z 1499.040,A 0.000,B 0.000,C 90.000,E1 43.095} C_DIS
LIN {X 0.396,Y -595.371,Z 1499.032,A 0.000,B 0.000,C 90.000,E1 41.757} C_DIS
LIN {X 0.153,Y -594.558,Z 1499.028,A 0.000,B 0.000,C 90.000,E1 40.987} C_DIS
LIN {X 0.086,Y -592.612,Z 1499.019,A 0.000,B 0.000,C 90.000,E1 39.402} C_DIS
LIN {X -0.320,Y -591.818,Z 1499.016,A 0.000,B 0.000,C 90.000,E1 38.910} C_DIS
LIN {X 0.062,Y -590.087,Z 1499.010,A 0.000,B 0.000,C 90.000,E1 37.810} C_DIS
LIN {X 0.058,Y -587.962,Z 1499.004,A 0.000,B 0.000,C 90.000,E1 36.744} C_DIS
LIN {X 0.178,Y -586.115,Z 1499.000,A 0.000,B 0.000,C 90.000,E1 35.931} C_DIS
LIN {X -0.071,Y -584.149,Z 1498.995,A 0.000,B 0.000,C 90.000,E1 35.152} C_DIS
LIN {X 0.138,Y -581.868,Z 1498.991,A 0.000,B 0.000,C 90.000,E1 34.326} C_DIS
LIN {X 0.168,Y -578.390,Z 1498.985,A 0.000,B 0.000,C 90.000,E1 33.245} C_DIS
LIN {X -0.316,Y -576.325,Z 1498.982,A 0.000,B 0.000,C 90.000,E1 32.752} C_DIS
LIN {X -0.248,Y -574.482,Z 1498.980,A 0.000,B 0.000,C 90.000,E1 32.339} C_DIS
LIN {X -0.191,Y -572.282,Z 1498.977,A 0.000,B 0.000,C 90.000,E1 31.926} C_DIS
LIN {X 0.334,Y -569.515,Z 1498.975,A 0.000,B 0.000,C 90.000,E1 31.465} C_DIS
LIN {X 0.157,Y -567.184,Z 1498.974,A 0.000,B 0.000,C 90.000,E1 31.209} C_DIS
LIN {X -0.189,Y -565.024,Z 1498.972,A 0.000,B 0.000,C 90.000,E1 31.052} C_DIS
LIN {X 0.031,Y -563.295,Z 1498.972,A 0.000,B 0.000,C 90.000,E1 30.924} C_DIS
LIN {X 0.104,Y -561.886,Z 1498.972,A 0.000,B 0.000,C 90.000,E1 30.875} C_DIS
LIN {X 0.049,Y -391.938,Z 1498.972,A 0.000,B 0.000,C 90.000,E1 30.875} C_DIS
LIN {X 0.086,Y -384.507,Z 1498.946,A 0.000,B 0.000,C 90.000,E1 26.181} C_DIS
LIN {X -0.114,Y -382.778,Z 1498.938,A 0.000,B 0.000,C 90.000,E1 24.771} C_DIS
LIN {X -0.158,Y -376.090,Z 1498.911,A 0.000,B 0.000,C 90.000,E1 20.066} C_DIS
LIN {X 0.183,Y -373.622,Z 1498.897,A 0.000,B 0.000,C 90.000,E1 17.457} C_DIS
LIN {X -0.144,Y -368.023,Z 1498.869,A 0.000,B 0.000,C 90.000,E1 12.355} C_DIS
LIN {X 0.089,Y -366.317,Z 1498.854,A 0.000,B 0.000,C 90.000,E1 9.726} C_DIS
LIN {X -0.032,Y -361.707,Z 1498.821,A 0.000,B 0.000,C 90.000,E1 3.784} C_DIS
LIN {X 0.049,Y -360.909,Z 1498.802,A 0.000,B 0.000,C 90.000,E1 0.401} C_DIS
LIN {X 0.137,Y -360.684,Z 1498.799,A 0.000,B 0.000,C 90.000,E1 359.771} C_DIS
LIN {X -0.053,Y -359.426,Z 1498.770,A 0.000,B 0.000,C 90.000,E1 354.546} C_DIS
LIN {X 0.070,Y -358.890,Z 1498.759,A 0.000,B 0.000,C 90.000,E1 352.648} C_DIS
LIN {X -0.020,Y -359.563,Z 1498.726,A 0.000,B 0.000,C 90.000,E1 346.645} C_DIS
LIN {X 0.001,Y -361.801,Z 1498.684,A 0.000,B 0.000,C 90.000,E1 339.135} C_DIS
LIN {X -0.154,Y -362.053,Z 1498.680,A 0.000,B 0.000,C 90.000,E1 338.411} C_DIS
LIN {X 0.189,Y -365.980,Z 1498.643,A 0.000,B 0.000,C 90.000,E1 331.641} C_DIS
LIN {X 0.029,Y -366.387,Z 1498.639,A 0.000,B 0.000,C 90.000,E1 330.923} C_DIS
LIN {X -0.031,Y -371.355,Z 1498.604,A 0.000,B 0.000,C 90.000,E1 324.642} C_DIS
LIN {X -0.043,Y -371.766,Z 1498.602,A 0.000,B 0.000,C 90.000,E1 324.276} C_DIS
LIN {X 0.013,Y -377.358,Z 1498.567,A 0.000,B 0.000,C 90.000,E1 318.038} C_DIS
LIN {X 0.012,Y -378.235,Z 1498.563,A 0.000,B 0.000,C 90.000,E1 317.310} C_DIS
LIN {X 0.002,Y -383.940,Z 1498.531,A 0.000,B 0.000,C 90.000,E1 311.515} C_DIS
LIN {X 0.088,Y -384.893,Z 1498.527,A 0.000,B 0.000,C 90.000,E1 310.782} C_DIS
LIN {X 0.262,Y -390.610,Z 1498.495,A 0.000,B 0.000,C 90.000,E1 305.025} C_DIS
LIN {X 0.106,Y -391.104,Z 1498.493,A 0.000,B 0.000,C 90.000,E1 304.692} C_DIS
LIN {X 0.022,Y -391.648,Z 1498.489,A 0.000,B 0.000,C 90.000,E1 303.992} C_DIS
LIN {X -0.080,Y -396.825,Z 1498.459,A 0.000,B 0.000,C 90.000,E1 298.693} C_DIS
LIN {X -0.210,Y -397.120,Z 1498.457,A 0.000,B 0.000,C 90.000,E1 298.359} C_DIS
LIN {X -0.055,Y -401.597,Z 1498.426,A 0.000,B 0.000,C 90.000,E1 292.717} C_DIS
LIN {X 0.222,Y -404.659,Z 1498.395,A 0.000,B 0.000,C 90.000,E1 287.094} C_DIS
END
